  MoveL 1954 to (322.8, 56.16, -151.37) mm, rotated rx -179.9 ry 0 rz -90 deg; joints [37.248, -66.49, 102.161, -126.692, 48.997, 139.557]
  MoveL 1955 to (320.86, 56.08, -150.36) mm, rotated rx -179.9 ry 0 rz -90 deg; joints [37.212, -66.609, 102.338, -126.77, 49.008, 139.643]
  MoveL 1956 to (318.69, 56.01, -150.1) mm, rotated rx -179.9 ry 0 rz -90 deg; joints [37.149, -66.699, 102.475, -126.865, 48.995, 139.733]
  MoveL 1957 to (316.57, 55.93, -150.63) mm, rotated rx -179.9 ry 0 rz -90 deg; joints [37.069, -66.749, 102.554, -126.966, 48.961, 139.816]
  MoveL 1958 to (314.78, 55.85, -151.88) mm, rotated rx -179.9 ry 0 rz -90 deg; joints [36.982, -66.751, 102.565, -127.061, 48.91, 139.882]
  MoveL 1959 to (313.55, 55.78, -153.69) mm, rotated rx -179.9 ry 0 rz -90 deg; joints [36.899, -66.705, 102.507, -127.136, 48.849, 139.923]
  MoveL 1960 to (313.04, 55.7, -155.81) mm, rotated rx -179.9 ry 0 rz -90 deg; joints [36.832, -66.617, 102.388, -127.182, 48.787, 139.933]
  MoveL 1961 to (313.33, 55.62, -157.98) mm, rotated rx -179.9 ry 0 rz -90 deg; joints [36.789, -66.498, 102.224, -127.194, 48.732, 139.913]
  MoveL 1962 to (314.37, 55.55, -159.9) mm, rotated rx -179.9 ry 0 rz -90 deg; joints [36.777, -66.364, 102.036, -127.17, 48.692, 139.866]
  MoveL 1963 to (316.03, 55.47, -161.33) mm, rotated rx -179.9 ry 0 rz -90 deg; joints [36.795, -66.231, 101.851, -127.114, 48.672, 139.797]
  MoveL 1964 to (318.09, 55.39, -162.07) mm, rotated rx -179.9 ry 0 rz -90 deg; joints [36.843, -66.118, 101.691, -127.033, 48.675, 139.717]
  MoveL 1965 to (320.27, 55.32, -162.03) mm, rotated rx -179.9 ry 0 rz -90 deg; joints [36.913, -66.038, 101.58, -126.94, 48.702, 139.638]
  MoveL 1966 to (322.3, 55.24, -161.21) mm, rotated rx -179.9 ry 0 rz -90 deg; joints [36.997, -66.001, 101.531, -126.847, 48.749, 139.571]
  MoveL 1967 to (323.9, 55.16, -159.73) mm, rotated rx -179.9 ry 0 rz -90 deg; joints [37.083, -66.013, 101.552, -126.766, 48.811, 139.524]
  MoveL 1968 to (324.87, 55.09, -157.77) mm, rotated rx -179.9 ry 0 rz -90 deg; joints [37.161, -66.071, 101.64, -126.709, 48.879, 139.506]
  MoveL 1969 to (325.08, 55.01, -155.59) mm, rotated rx -179.9 ry 0 rz -90 deg; joints [37.219, -66.168, 101.784, -126.683, 48.946, 139.518]
  MoveL 1970 to (324.49, 54.93, -153.48) mm, rotated rx -179.9 ry 0 rz -90 deg; joints [37.252, -66.29, 101.965, -126.692, 49.002, 139.56]
  MoveL 1971 to (323.2, 54.86, -151.72) mm, rotated rx -179.9 ry 0 rz -90 deg; joints [37.253, -66.421, 102.16, -126.735, 49.041, 139.627]
  MoveL 1972 to (321.36, 54.78, -150.54) mm, rotated rx -179.9 ry 0 rz -90 deg; joints [37.224, -66.544, 102.344, -126.807, 49.058, 139.71]
  MoveL 1973 to (319.22, 54.7, -150.09) mm, rotated rx -179.9 ry 0 rz -90 deg; joints [37.167, -66.643, 102.493, -126.899, 49.051, 139.8]
  MoveL 1974 to (317.06, 54.63, -150.43) mm, rotated rx -179.9 ry 0 rz -90 deg; joints [37.09, -66.703, 102.587, -127, 49.022, 139.886]
  MoveL 1975 to (315.17, 54.55, -151.52) mm, rotated rx -179.9 ry 0 rz -90 deg; joints [37.004, -66.717, 102.615, -127.097, 48.975, 139.956]
  MoveL 1976 to (313.78, 54.47, -153.21) mm, rotated rx -179.9 ry 0 rz -90 deg; joints [36.919, -66.682, 102.573, -127.178, 48.916, 140.004]
  MoveL 1977 to (313.09, 54.4, -155.28) mm, rotated rx -179.9 ry 0 rz -90 deg; joints [36.847, -66.604, 102.468, -127.232, 48.853, 140.022]
  MoveL 1978 to (313.19, 54.32, -157.47) mm, rotated rx -179.9 ry 0 rz -90 deg; joints [36.798, -66.491, 102.313, -127.252, 48.796, 140.009]
  MoveL 1979 to (314.06, 54.24, -159.47) mm, rotated rx -179.9 ry 0 rz -90 deg; joints [36.778, -66.359, 102.129, -127.237, 48.751, 139.968]
  MoveL 1980 to (315.58, 54.16, -161.04) mm, rotated rx -179.9 ry 0 rz -90 deg; joints [36.789, -66.224, 101.94, -127.188, 48.726, 139.903]
  MoveL 1981 to (317.56, 54.09, -161.96) mm, rotated rx -179.9 ry 0 rz -90 deg; joints [36.83, -66.105, 101.772, -127.112, 48.723, 139.826]
  MoveL 1982 to (319.74, 54.01, -162.11) mm, rotated rx -179.9 ry 0 rz -90 deg; joints [36.895, -66.016, 101.648, -127.021, 48.744, 139.745]
  MoveL 1983 to (321.84, 53.93, -161.48) mm, rotated rx -179.9 ry 0 rz -90 deg; joints [36.977, -65.968, 101.583, -126.927, 48.787, 139.674]
  MoveL 1984 to (323.57, 53.86, -160.14) mm, rotated rx -179.9 ry 0 rz -90 deg; joints [37.063, -65.968, 101.587, -126.842, 48.845, 139.622]
  MoveL 1985 to (324.7, 53.78, -158.27) mm, rotated rx -179.9 ry 0 rz -90 deg; joints [37.144, -66.016, 101.659, -126.778, 48.913, 139.596]
  MoveL 1986 to (325.1, 53.7, -156.12) mm, rotated rx -179.9 ry 0 rz -90 deg; joints [37.208, -66.104, 101.791, -126.744, 48.981, 139.601]
  MoveL 1987 to (324.71, 53.63, -153.97) mm, rotated rx -179.9 ry 0 rz -90 deg; joints [37.247, -66.221, 101.965, -126.744, 49.04, 139.636]
  MoveL 1988 to (323.57, 53.55, -152.1) mm, rotated rx -179.9 ry 0 rz -90 deg; joints [37.256, -66.352, 102.159, -126.779, 49.084, 139.698]
  MoveL 1989 to (321.85, 53.47, -150.76) mm, rotated rx -179.9 ry 0 rz -90 deg; joints [37.234, -66.478, 102.348, -126.845, 49.107, 139.778]
  MoveL 1990 to (319.75, 53.4, -150.12) mm, rotated rx -179.9 ry 0 rz -90 deg; joints [37.183, -66.584, 102.507, -126.933, 49.106, 139.867]
  MoveL 1991 to (317.57, 53.32, -150.27) mm, rotated rx -179.9 ry 0 rz -90 deg; joints [37.111, -66.654, 102.616, -127.033, 49.082, 139.954]
  MoveL 1992 to (315.59, 53.24, -151.19) mm, rotated rx -179.9 ry 0 rz -90 deg; joints [37.025, -66.68, 102.66, -127.132, 49.039, 140.03]
  MoveL 1993 to (314.06, 53.17, -152.75) mm, rotated rx -179.9 ry 0 rz -90 deg; joints [36.939, -66.657, 102.635, -127.218, 48.982, 140.083]
  MoveL 1994 to (313.19, 53.09, -154.76) mm, rotated rx -179.9 ry 0 rz -90 deg; joints [36.863, -66.588, 102.544, -127.279, 48.919, 140.109]
  MoveL 1995 to (313.09, 53.01, -156.94) mm, rotated rx -179.9 ry 0 rz -90 deg; joints [36.808, -66.483, 102.4, -127.308, 48.86, 140.104]
  MoveL 1996 to (313.78, 52.94, -159.02) mm, rotated rx -179.9 ry 0 rz -90 deg; joints [36.78, -66.354, 102.22, -127.302, 48.812, 140.069]
  MoveL 1997 to (315.16, 52.86, -160.71) mm, rotated rx -179.9 ry 0 rz -90 deg; joints [36.784, -66.218, 102.031, -127.26, 48.781, 140.009]
  MoveL 1998 to (317.05, 52.78, -161.8) mm, rotated rx -179.9 ry 0 rz -90 deg; joints [36.818, -66.094, 101.856, -127.19, 48.773, 139.933]
  MoveL 1999 to (319.21, 52.71, -162.15) mm, rotated rx -179.9 ry 0 rz -90 deg; joints [36.878, -65.996, 101.719, -127.102, 48.788, 139.853]
  MoveL 2000 to (321.35, 52.63, -161.7) mm, rotated rx -179.9 ry 0 rz -90 deg; joints [36.957, -65.938, 101.638, -127.007, 48.825, 139.778]
  MoveL 2001 to (323.19, 52.55, -160.52) mm, rotated rx -179.9 ry 0 rz -90 deg; joints [37.043, -65.926, 101.625, -126.919, 48.881, 139.72]
  MoveL 2002 to (324.49, 52.48, -158.76) mm, rotated rx -179.9 ry 0 rz -90 deg; joints [37.126, -65.962, 101.681, -126.849, 48.947, 139.688]
  MoveL 2003 to (325.08, 52.4, -156.65) mm, rotated rx -179.9 ry 0 rz -90 deg; joints [37.195, -66.041, 101.8, -126.807, 49.015, 139.685]
  MoveL 2004 to (324.87, 52.32, -154.48) mm, rotated rx -179.9 ry 0 rz -90 deg; joints [37.241, -66.153, 101.966, -126.799, 49.078, 139.714]
  MoveL 2005 to (323.91, 52.25, -152.52) mm, rotated rx -179.9 ry 0 rz -90 deg; joints [37.258, -66.282, 102.158, -126.825, 49.126, 139.769]
  MoveL 2006 to (322.31, 52.17, -151.03) mm, rotated rx -179.9 ry 0 rz -90 deg; joints [37.243, -66.411, 102.35, -126.884, 49.154, 139.845]
  MoveL 2007 to (320.28, 52.09, -150.21) mm, rotated rx -179.9 ry 0 rz -90 deg; joints [37.199, -66.523, 102.518, -126.967, 49.159, 139.933]
  MoveL 2008 to (318.09, 52.02, -150.16) mm, rotated rx -179.9 ry 0 rz -90 deg; joints [37.13, -66.603, 102.641, -127.065, 49.141, 140.022]
  MoveL 2009 to (316.04, 51.94, -150.9) mm, rotated rx -179.9 ry 0 rz -90 deg; joints [37.047, -66.64, 102.702, -127.166, 49.102, 140.101]
  MoveL 2010 to (314.38, 51.86, -152.32) mm, rotated rx -179.9 ry 0 rz -90 deg; joints [36.96, -66.629, 102.693, -127.256, 49.048, 140.161]
  MoveL 2011 to (313.33, 51.79, -154.25) mm, rotated rx -179.9 ry 0 rz -90 deg; joints [36.881, -66.57, 102.618, -127.325, 48.986, 140.194]
  MoveL 2012 to (313.04, 51.71, -156.41) mm, rotated rx -179.9 ry 0 rz -90 deg; joints [36.82, -66.473, 102.484, -127.362, 48.925, 140.196]
  MoveL 2013 to (313.54, 51.63, -158.54) mm, rotated rx -179.9 ry 0 rz -90 deg; joints [36.785, -66.348, 102.312, -127.364, 48.873, 140.168]
  MoveL 2014 to (314.77, 51.56, -160.35) mm, rotated rx -179.9 ry 0 rz -90 deg; joints [36.781, -66.213, 102.122, -127.331, 48.838, 140.113]
  MoveL 2015 to (316.56, 51.48, -161.6) mm, rotated rx -179.9 ry 0 rz -90 deg; joints [36.808, -66.084, 101.941, -127.267, 48.824, 140.041]
  MoveL 2016 to (318.68, 51.4, -162.14) mm, rotated rx -179.9 ry 0 rz -90 deg; joints [36.862, -65.979, 101.793, -127.182, 48.833, 139.96]
  MoveL 2017 to (320.85, 51.32, -161.88) mm, rotated rx -179.9 ry 0 rz -90 deg; joints [36.937, -65.91, 101.698, -127.088, 48.865, 139.883]
  MoveL 2018 to (322.79, 51.25, -160.87) mm, rotated rx -179.9 ry 0 rz -90 deg; joints [37.023, -65.887, 101.668, -126.997, 48.917, 139.821]
  MoveL 2019 to (324.24, 51.17, -159.23) mm, rotated rx -179.9 ry 0 rz -90 deg; joints [37.107, -65.911, 101.707, -126.921, 48.981, 139.781]
  MoveL 2020 to (325.01, 51.09, -157.18) mm, rotated rx -179.9 ry 0 rz -90 deg; joints [37.181, -65.981, 101.812, -126.872, 49.049, 139.771]
  MoveL 2021 to (325, 51.02, -155) mm, rotated rx -179.9 ry 0 rz -90 deg; joints [37.233, -66.086, 101.968, -126.855, 49.114, 139.792]
  MoveL 2022 to (324.21, 50.94, -152.96) mm, rotated rx -179.9 ry 0 rz -90 deg; joints [37.257, -66.212, 102.156, -126.873, 49.167, 139.842]
  MoveL 2023 to (322.74, 50.86, -151.33) mm, rotated rx -179.9 ry 0 rz -90 deg; joints [37.25, -66.342, 102.35, -126.924, 49.2, 139.914]
  MoveL 2024 to (320.8, 50.79, -150.34) mm, rotated rx -179.9 ry 0 rz -90 deg; joints [37.213, -66.46, 102.526, -127.002, 49.211, 140]
  MoveL 2025 to (318.62, 50.71, -150.1) mm, rotated rx -179.9 ry 0 rz -90 deg; joints [37.149, -66.549, 102.662, -127.098, 49.199, 140.089]
  MoveL 2026 to (316.51, 50.63, -150.65) mm, rotated rx -179.9 ry 0 rz -90 deg; joints [37.069, -66.597, 102.739, -127.199, 49.164, 140.172]
  MoveL 2027 to (314.73, 50.56, -151.93) mm, rotated rx -179.9 ry 0 rz -90 deg; joints [36.982, -66.597, 102.748, -127.293, 49.113, 140.237]
  MoveL 2028 to (313.52, 50.48, -153.75) mm, rotated rx -179.9 ry 0 rz -90 deg; joints [36.899, -66.55, 102.687, -127.368, 49.053, 140.276]
  MoveL 2029 to (313.04, 50.4, -155.88) mm, rotated rx -179.9 ry 0 rz -90 deg; joints [36.833, -66.461, 102.567, -127.414, 48.991, 140.286]
  MoveL 2030 to (313.35, 50.33, -158.04) mm, rotated rx -179.9 ry 0 rz -90 deg; joints [36.791, -66.342, 102.401, -127.424, 48.936, 140.265]
  MoveL 2031 to (314.41, 50.25, -159.95) mm, rotated rx -179.9 ry 0 rz -90 deg; joints [36.78, -66.207, 102.214, -127.399, 48.896, 140.217]
  MoveL 2032 to (316.09, 50.17, -161.36) mm, rotated rx -179.9 ry 0 rz -90 deg; joints [36.799, -66.076, 102.028, -127.342, 48.876, 140.147]
  MoveL 2033 to (318.15, 50.1, -162.08) mm, rotated rx -179.9 ry 0 rz -90 deg; joints [36.848, -65.963, 101.87, -127.262, 48.88, 140.068]
  MoveL 2034 to (320.34, 50.02, -162.02) mm, rotated rx -179.9 ry 0 rz -90 deg; joints [36.918, -65.885, 101.761, -127.168, 48.906, 139.989]
  MoveL 2035 to (322.36, 49.94, -161.18) mm, rotated rx -179.9 ry 0 rz -90 deg; joints [37.002, -65.85, 101.714, -127.075, 48.953, 139.922]
  MoveL 2036 to (323.94, 49.87, -159.67) mm, rotated rx -179.9 ry 0 rz -90 deg; joints [37.088, -65.863, 101.737, -126.995, 49.015, 139.876]
  MoveL 2037 to (324.89, 49.79, -157.7) mm, rotated rx -179.9 ry 0 rz -90 deg; joints [37.165, -65.922, 101.827, -126.938, 49.083, 139.859]
  MoveL 2038 to (325.07, 49.71, -155.52) mm, rotated rx -179.9 ry 0 rz -90 deg; joints [37.223, -66.02, 101.972, -126.913, 49.15, 139.873]
  MoveL 2039 to (324.47, 49.64, -153.42) mm, rotated rx -179.9 ry 0 rz -90 deg; joints [37.255, -66.142, 102.154, -126.922, 49.206, 139.915]
  MoveL 2040 to (323.15, 49.56, -151.68) mm, rotated rx -179.9 ry 0 rz -90 deg; joints [37.256, -66.273, 102.349, -126.966, 49.245, 139.983]
  MoveL 2041 to (321.3, 49.48, -150.51) mm, rotated rx -179.9 ry 0 rz -90 deg; joints [37.225, -66.395, 102.532, -127.039, 49.262, 140.066]
  MoveL 2042 to (319.16, 49.41, -150.09) mm, rotated rx -179.9 ry 0 rz -90 deg; joints [37.167, -66.492, 102.679, -127.131, 49.255, 140.156]
  MoveL 2043 to (317, 49.33, -150.45) mm, rotated rx -179.9 ry 0 rz -90 deg; joints [37.09, -66.551, 102.772, -127.232, 49.226, 140.241]
  MoveL 2044 to (315.12, 49.25, -151.56) mm, rotated rx -179.9 ry 0 rz -90 deg; joints [37.004, -66.563, 102.797, -127.329, 49.178, 140.311]
  MoveL 2045 to (313.75, 49.18, -153.27) mm, rotated rx -179.9 ry 0 rz -90 deg; joints [36.919, -66.527, 102.754, -127.409, 49.119, 140.357]
  MoveL 2046 to (313.08, 49.1, -155.35) mm, rotated rx -179.9 ry 0 rz -90 deg; joints [36.848, -66.448, 102.646, -127.463, 49.057, 140.375]
  MoveL 2047 to (313.2, 49.02, -157.53) mm, rotated rx -179.9 ry 0 rz -90 deg; joints [36.799, -66.334, 102.49, -127.482, 49, 140.361]
  MoveL 2048 to (314.09, 48.94, -159.53) mm, rotated rx -179.9 ry 0 rz -90 deg; joints [36.78, -66.202, 102.305, -127.466, 48.955, 140.318]
  MoveL 2049 to (315.64, 48.87, -161.08) mm, rotated rx -179.9 ry 0 rz -90 deg; joints [36.792, -66.068, 102.117, -127.416, 48.93, 140.253]
  MoveL 2050 to (317.63, 48.79, -161.98) mm, rotated rx -179.9 ry 0 rz -90 deg; joints [36.834, -65.95, 101.95, -127.34, 48.928, 140.175]
  MoveL 2051 to (319.81, 48.71, -162.1) mm, rotated rx -179.9 ry 0 rz -90 deg; joints [36.9, -65.862, 101.827, -127.249, 48.949, 140.095]
  MoveL 2052 to (321.9, 48.64, -161.45) mm, rotated rx -179.9 ry 0 rz -90 deg; joints [36.982, -65.816, 101.764, -127.154, 48.991, 140.024]
  MoveL 2053 to (323.61, 48.56, -160.09) mm, rotated rx -179.9 ry 0 rz -90 deg; joints [37.068, -65.817, 101.77, -127.07, 49.05, 139.973]
  MoveL 2054 to (324.73, 48.48, -158.21) mm, rotated rx -179.9 ry 0 rz -90 deg; joints [37.149, -65.866, 101.845, -127.006, 49.117, 139.948]
  MoveL 2055 to (325.1, 48.41, -156.06) mm, rotated rx -179.9 ry 0 rz -90 deg; joints [37.212, -65.955, 101.978, -126.973, 49.185, 139.954]
  MoveL 2056 to (324.68, 48.33, -153.91) mm, rotated rx -179.9 ry 0 rz -90 deg; joints [37.251, -66.073, 102.153, -126.974, 49.245, 139.99]
  MoveL 2057 to (323.53, 48.25, -152.05) mm, rotated rx -179.9 ry 0 rz -90 deg; joints [37.259, -66.203, 102.348, -127.01, 49.288, 140.052]
  MoveL 2058 to (321.79, 48.18, -150.73) mm, rotated rx -179.9 ry 0 rz -90 deg; joints [37.236, -66.329, 102.536, -127.076, 49.311, 140.133]
  MoveL 2059 to (319.69, 48.1, -150.12) mm, rotated rx -179.9 ry 0 rz -90 deg; joints [37.184, -66.433, 102.693, -127.164, 49.31, 140.222]
  MoveL 2060 to (317.51, 48.02, -150.29) mm, rotated rx -179.9 ry 0 rz -90 deg; joints [37.111, -66.502, 102.8, -127.265, 49.286, 140.309]
  MoveL 2061 to (315.53, 47.95, -151.23) mm, rotated rx -179.9 ry 0 rz -90 deg; joints [37.025, -66.526, 102.843, -127.364, 49.242, 140.384]
  MoveL 2062 to (314.02, 47.87, -152.81) mm, rotated rx -179.9 ry 0 rz -90 deg; joints [36.939, -66.502, 102.816, -127.449, 49.185, 140.436]
  MoveL 2063 to (313.18, 47.79, -154.82) mm, rotated rx -179.9 ry 0 rz -90 deg; joints [36.864, -66.432, 102.723, -127.51, 49.123, 140.461]
  MoveL 2064 to (313.1, 47.72, -157.01) mm, rotated rx -179.9 ry 0 rz -90 deg; joints [36.809, -66.326, 102.577, -127.538, 49.064, 140.455]
  MoveL 2065 to (313.81, 47.64, -159.08) mm, rotated rx -179.9 ry 0 rz -90 deg; joints [36.783, -66.197, 102.397, -127.53, 49.016, 140.419]
  MoveL 2066 to (315.21, 47.56, -160.76) mm, rotated rx -179.9 ry 0 rz -90 deg; joints [36.787, -66.061, 102.207, -127.488, 48.986, 140.358]
  MoveL 2067 to (317.12, 47.49, -161.83) mm, rotated rx -179.9 ry 0 rz -90 deg; joints [36.822, -65.938, 102.033, -127.418, 48.977, 140.282]
  MoveL 2068 to (319.28, 47.41, -162.15) mm, rotated rx -179.9 ry 0 rz -90 deg; joints [36.883, -65.841, 101.897, -127.329, 48.993, 140.202]
  MoveL 2069 to (321.42, 47.33, -161.67) mm, rotated rx -179.9 ry 0 rz -90 deg; joints [36.962, -65.784, 101.819, -127.234, 49.03, 140.128]
  MoveL 2070 to (323.24, 47.26, -160.47) mm, rotated rx -179.9 ry 0 rz -90 deg; joints [37.048, -65.774, 101.808, -127.146, 49.085, 140.071]
  MoveL 2071 to (324.52, 47.18, -158.7) mm, rotated rx -179.9 ry 0 rz -90 deg; joints [37.131, -65.812, 101.866, -127.076, 49.151, 140.039]
  MoveL 2072 to (325.08, 47.1, -156.59) mm, rotated rx -179.9 ry 0 rz -90 deg; joints [37.2, -65.892, 101.987, -127.035, 49.22, 140.038]
  MoveL 2073 to (324.85, 47.03, -154.41) mm, rotated rx -179.9 ry 0 rz -90 deg; joints [37.245, -66.004, 102.154, -127.027, 49.282, 140.067]
  MoveL 2074 to (323.87, 46.95, -152.46) mm, rotated rx -179.9 ry 0 rz -90 deg; joints [37.261, -66.133, 102.345, -127.055, 49.33, 140.123]
  MoveL 2075 to (322.25, 46.87, -150.99) mm, rotated rx -179.9 ry 0 rz -90 deg; joints [37.245, -66.261, 102.537, -127.114, 49.359, 140.2]
  MoveL 2076 to (320.21, 46.8, -150.19) mm, rotated rx -179.9 ry 0 rz -90 deg; joints [37.2, -66.372, 102.705, -127.198, 49.363, 140.288]
  MoveL 2077 to (318.03, 46.72, -150.18) mm, rotated rx -179.9 ry 0 rz -90 deg; joints [37.131, -66.451, 102.825, -127.297, 49.345, 140.377]
  MoveL 2078 to (315.98, 46.64, -150.94) mm, rotated rx -179.9 ry 0 rz -90 deg; joints [37.047, -66.486, 102.884, -127.397, 49.306, 140.455]
  MoveL 2079 to (314.34, 46.57, -152.38) mm, rotated rx -179.9 ry 0 rz -90 deg; joints [36.96, -66.473, 102.874, -127.487, 49.252, 140.514]
  MoveL 2080 to (313.31, 46.49, -154.31) mm, rotated rx -179.9 ry 0 rz -90 deg; joints [36.881, -66.414, 102.796, -127.555, 49.19, 140.545]
  MoveL 2081 to (313.05, 46.41, -156.48) mm, rotated rx -179.9 ry 0 rz -90 deg; joints [36.821, -66.315, 102.661, -127.591, 49.129, 140.547]
  MoveL 2082 to (313.57, 46.33, -158.6) mm, rotated rx -179.9 ry 0 rz -90 deg; joints [36.787, -66.19, 102.487, -127.592, 49.078, 140.517]
  MoveL 2083 to (314.82, 46.26, -160.4) mm, rotated rx -179.9 ry 0 rz -90 deg; joints [36.784, -66.055, 102.298, -127.558, 49.042, 140.462]
  MoveL 2084 to (316.62, 46.18, -161.63) mm, rotated rx -179.9 ry 0 rz -90 deg; joints [36.812, -65.927, 102.118, -127.494, 49.028, 140.389]
  MoveL 2085 to (318.75, 46.1, -162.14) mm, rotated rx -179.9 ry 0 rz -90 deg; joints [36.867, -65.823, 101.971, -127.408, 49.038, 140.309]
  MoveL 2086 to (320.92, 46.03, -161.86) mm, rotated rx -179.9 ry 0 rz -90 deg; joints [36.942, -65.756, 101.877, -127.314, 49.07, 140.232]
  MoveL 2087 to (322.84, 45.95, -160.82) mm, rotated rx -179.9 ry 0 rz -90 deg; joints [37.028, -65.734, 101.849, -127.223, 49.122, 140.17]
  MoveL 2088 to (324.27, 45.87, -159.17) mm, rotated rx -179.9 ry 0 rz -90 deg; joints [37.113, -65.76, 101.891, -127.148, 49.186, 140.132]
  MoveL 2089 to (325.02, 45.8, -157.12) mm, rotated rx -179.9 ry 0 rz -90 deg; joints [37.185, -65.831, 101.998, -127.099, 49.254, 140.123]
  MoveL 2090 to (324.98, 45.72, -154.93) mm, rotated rx -179.9 ry 0 rz -90 deg; joints [37.237, -65.936, 102.155, -127.083, 49.319, 140.145]
  MoveL 2091 to (324.17, 45.64, -152.9) mm, rotated rx -179.9 ry 0 rz -90 deg; joints [37.26, -66.062, 102.343, -127.102, 49.371, 140.195]
  MoveL 2092 to (322.69, 45.57, -151.29) mm, rotated rx -179.9 ry 0 rz -90 deg; joints [37.252, -66.192, 102.537, -127.154, 49.405, 140.267]
  MoveL 2093 to (320.73, 45.49, -150.32) mm, rotated rx -179.9 ry 0 rz -90 deg; joints [37.214, -66.309, 102.713, -127.233, 49.416, 140.354]
  MoveL 2094 to (318.56, 45.41, -150.11) mm, rotated rx -179.9 ry 0 rz -90 deg; joints [37.15, -66.396, 102.846, -127.329, 49.403, 140.443]
  MoveL 2095 to (316.45, 45.34, -150.68) mm, rotated rx -179.9 ry 0 rz -90 deg; joints [37.069, -66.443, 102.921, -127.43, 49.368, 140.525]
  MoveL 2096 to (314.68, 45.26, -151.97) mm, rotated rx -179.9 ry 0 rz -90 deg; joints [36.982, -66.442, 102.928, -127.524, 49.317, 140.589]
  MoveL 2097 to (313.49, 45.18, -153.81) mm, rotated rx -179.9 ry 0 rz -90 deg; joints [36.9, -66.393, 102.866, -127.598, 49.257, 140.628]
  MoveL 2098 to (313.04, 45.11, -155.95) mm, rotated rx -179.9 ry 0 rz -90 deg; joints [36.834, -66.303, 102.743, -127.642, 49.195, 140.637]
  MoveL 2099 to (313.37, 45.03, -158.11) mm, rotated rx -179.9 ry 0 rz -90 deg; joints [36.793, -66.184, 102.577, -127.652, 49.141, 140.614]
  MoveL 2100 to (314.46, 44.95, -160.01) mm, rotated rx -179.9 ry 0 rz -90 deg; joints [36.782, -66.049, 102.389, -127.626, 49.101, 140.565]
  MoveL 2101 to (316.15, 44.88, -161.39) mm, rotated rx -179.9 ry 0 rz -90 deg; joints [36.803, -65.918, 102.204, -127.569, 49.081, 140.495]
  MoveL 2102 to (318.22, 44.8, -162.09) mm, rotated rx -179.9 ry 0 rz -90 deg; joints [36.852, -65.807, 102.047, -127.487, 49.085, 140.416]
  MoveL 2103 to (320.4, 44.72, -162) mm, rotated rx -179.9 ry 0 rz -90 deg; joints [36.923, -65.73, 101.939, -127.393, 49.112, 140.337]
  MoveL 2104 to (322.41, 44.65, -161.14) mm, rotated rx -179.9 ry 0 rz -90 deg; joints [37.008, -65.696, 101.895, -127.3, 49.159, 140.271]
  MoveL 2105 to (323.98, 44.57, -159.62) mm, rotated rx -179.9 ry 0 rz -90 deg; joints [37.093, -65.711, 101.92, -127.221, 49.22, 140.226]
  MoveL 2106 to (324.91, 44.49, -157.64) mm, rotated rx -179.9 ry 0 rz -90 deg; joints [37.17, -65.772, 102.011, -127.165, 49.288, 140.21]
  MoveL 2107 to (325.06, 44.42, -155.46) mm, rotated rx -179.9 ry 0 rz -90 deg; joints [37.228, -65.869, 102.158, -127.14, 49.355, 140.224]
  MoveL 2108 to (324.43, 44.34, -153.36) mm, rotated rx -179.9 ry 0 rz -90 deg; joints [37.258, -65.992, 102.341, -127.15, 49.411, 140.268]
  MoveL 2109 to (323.1, 44.26, -151.63) mm, rotated rx -179.9 ry 0 rz -90 deg; joints [37.258, -66.123, 102.536, -127.195, 49.45, 140.336]
  MoveL 2110 to (321.24, 44.19, -150.49) mm, rotated rx -179.9 ry 0 rz -90 deg; joints [37.226, -66.244, 102.718, -127.268, 49.466, 140.42]
  MoveL 2111 to (319.09, 44.11, -150.09) mm, rotated rx -179.9 ry 0 rz -90 deg; joints [37.168, -66.34, 102.864, -127.361, 49.459, 140.509]
  MoveL 2112 to (316.94, 44.03, -150.47) mm, rotated rx -179.9 ry 0 rz -90 deg; joints [37.09, -66.397, 102.954, -127.462, 49.43, 140.594]
  MoveL 2113 to (315.07, 43.96, -151.6) mm, rotated rx -179.9 ry 0 rz -90 deg; joints [37.004, -66.408, 102.978, -127.559, 49.382, 140.663]
  MoveL 2114 to (313.72, 43.88, -153.33) mm, rotated rx -179.9 ry 0 rz -90 deg; joints [36.919, -66.37, 102.932, -127.639, 49.323, 140.708]
  MoveL 2115 to (313.08, 43.8, -155.42) mm, rotated rx -179.9 ry 0 rz -90 deg; joints [36.849, -66.29, 102.823, -127.691, 49.261, 140.725]
  MoveL 2116 to (313.22, 43.72, -157.6) mm, rotated rx -179.9 ry 0 rz -90 deg; joints [36.801, -66.176, 102.665, -127.71, 49.204, 140.71]
  MoveL 2117 to (314.13, 43.65, -159.58) mm, rotated rx -179.9 ry 0 rz -90 deg; joints [36.783, -66.043, 102.48, -127.692, 49.16, 140.666]
  MoveL 2118 to (315.69, 43.57, -161.12) mm, rotated rx -179.9 ry 0 rz -90 deg; joints [36.796, -65.91, 102.292, -127.642, 49.135, 140.601]
  MoveL 2119 to (317.69, 43.49, -161.99) mm, rotated rx -179.9 ry 0 rz -90 deg; joints [36.839, -65.793, 102.126, -127.565, 49.133, 140.522]
  MoveL 2120 to (319.88, 43.42, -162.1) mm, rotated rx -179.9 ry 0 rz -90 deg; joints [36.905, -65.706, 102.005, -127.473, 49.154, 140.442]
  MoveL 2121 to (321.96, 43.34, -161.41) mm, rotated rx -179.9 ry 0 rz -90 deg; joints [36.987, -65.662, 101.944, -127.379, 49.197, 140.372]
  MoveL 2122 to (323.65, 43.26, -160.04) mm, rotated rx -179.9 ry 0 rz -90 deg; joints [37.074, -65.665, 101.952, -127.295, 49.255, 140.322]
  MoveL 2123 to (324.75, 43.19, -158.15) mm, rotated rx -179.9 ry 0 rz -90 deg; joints [37.154, -65.714, 102.028, -127.232, 49.323, 140.298]
  MoveL 2124 to (325.1, 43.11, -155.99) mm, rotated rx -179.9 ry 0 rz -90 deg; joints [37.217, -65.804, 102.163, -127.199, 49.39, 140.305]
  MoveL 2125 to (324.66, 43.03, -153.85) mm, rotated rx -179.9 ry 0 rz -90 deg; joints [37.254, -65.922, 102.339, -127.201, 49.45, 140.342]
  MoveL 2126 to (323.48, 42.96, -152) mm, rotated rx -179.9 ry 0 rz -90 deg; joints [37.261, -66.052, 102.534, -127.237, 49.493, 140.405]
  MoveL 2127 to (321.73, 42.88, -150.7) mm, rotated rx -179.9 ry 0 rz -90 deg; joints [37.237, -66.177, 102.721, -127.304, 49.516, 140.486]
  MoveL 2128 to (319.62, 42.8, -150.11) mm, rotated rx -179.9 ry 0 rz -90 deg; joints [37.185, -66.28, 102.878, -127.393, 49.514, 140.575]
  MoveL 2129 to (317.44, 42.73, -150.31) mm, rotated rx -179.9 ry 0 rz -90 deg; joints [37.111, -66.348, 102.983, -127.494, 49.49, 140.661]
  MoveL 2130 to (315.48, 42.65, -151.27) mm, rotated rx -179.9 ry 0 rz -90 deg; joints [37.025, -66.37, 103.023, -127.593, 49.447, 140.735]
  MoveL 2131 to (313.99, 42.57, -152.87) mm, rotated rx -179.9 ry 0 rz -90 deg; joints [36.94, -66.344, 102.994, -127.678, 49.39, 140.787]
  MoveL 2132 to (313.16, 42.5, -154.89) mm, rotated rx -179.9 ry 0 rz -90 deg; joints [36.865, -66.274, 102.899, -127.738, 49.328, 140.811]
  MoveL 2133 to (313.11, 42.42, -157.08) mm, rotated rx -179.9 ry 0 rz -90 deg; joints [36.811, -66.167, 102.752, -127.765, 49.269, 140.803]
  MoveL 2134 to (313.84, 42.34, -159.14) mm, rotated rx -179.9 ry 0 rz -90 deg; joints [36.785, -66.037, 102.571, -127.756, 49.221, 140.766]
  MoveL 2135 to (315.26, 42.27, -160.8) mm, rotated rx -179.9 ry 0 rz -90 deg; joints [36.79, -65.903, 102.381, -127.713, 49.191, 140.705]
  MoveL 2136 to (317.18, 42.19, -161.85) mm, rotated rx -179.9 ry 0 rz -90 deg; joints [36.826, -65.78, 102.208, -127.642, 49.183, 140.629]
  MoveL 2137 to (319.35, 42.11, -162.14) mm, rotated rx -179.9 ry 0 rz -90 deg; joints [36.888, -65.685, 102.074, -127.553, 49.198, 140.548]
  MoveL 2138 to (321.48, 42.04, -161.65) mm, rotated rx -179.9 ry 0 rz -90 deg; joints [36.967, -65.629, 101.997, -127.458, 49.236, 140.475]
  MoveL 2139 to (323.29, 41.96, -160.43) mm, rotated rx -179.9 ry 0 rz -90 deg; joints [37.054, -65.621, 101.988, -127.37, 49.291, 140.419]
  MoveL 2140 to (324.55, 41.88, -158.64) mm, rotated rx -179.9 ry 0 rz -90 deg; joints [37.136, -65.66, 102.049, -127.301, 49.357, 140.388]
  MoveL 2141 to (325.09, 41.81, -156.52) mm, rotated rx -179.9 ry 0 rz -90 deg; joints [37.204, -65.741, 102.171, -127.26, 49.425, 140.388]
  MoveL 2142 to (324.84, 41.73, -154.35) mm, rotated rx -179.9 ry 0 rz -90 deg; joints [37.248, -65.853, 102.339, -127.254, 49.487, 140.418]
  MoveL 2143 to (323.83, 41.65, -152.41) mm, rotated rx -179.9 ry 0 rz -90 deg; joints [37.263, -65.982, 102.531, -127.282, 49.535, 140.475]
  MoveL 2144 to (322.19, 41.58, -150.96) mm, rotated rx -179.9 ry 0 rz -90 deg; joints [37.247, -66.109, 102.723, -127.342, 49.564, 140.552]
  MoveL 2145 to (320.15, 41.5, -150.18) mm, rotated rx -179.9 ry 0 rz -90 deg; joints [37.201, -66.219, 102.889, -127.426, 49.568, 140.64]
  MoveL 2146 to (317.96, 41.42, -150.19) mm, rotated rx -179.9 ry 0 rz -90 deg; joints [37.131, -66.296, 103.008, -127.525, 49.55, 140.728]
  MoveL 2147 to (315.92, 41.35, -150.97) mm, rotated rx -179.9 ry 0 rz -90 deg; joints [37.047, -66.33, 103.065, -127.626, 49.51, 140.806]
  MoveL 2148 to (314.29, 41.27, -152.43) mm, rotated rx -179.9 ry 0 rz -90 deg; joints [36.96, -66.316, 103.052, -127.715, 49.456, 140.864]
  MoveL 2149 to (313.29, 41.19, -154.37) mm, rotated rx -179.9 ry 0 rz -90 deg; joints [36.882, -66.255, 102.972, -127.782, 49.395, 140.895]
  MoveL 2150 to (313.05, 41.11, -156.55) mm, rotated rx -179.9 ry 0 rz -90 deg; joints [36.822, -66.156, 102.836, -127.818, 49.334, 140.895]
  MoveL 2151 to (313.6, 41.04, -158.66) mm, rotated rx -179.9 ry 0 rz -90 deg; joints [36.789, -66.031, 102.661, -127.818, 49.283, 140.865]
  MoveL 2152 to (314.87, 40.96, -160.45) mm, rotated rx -179.9 ry 0 rz -90 deg; joints [36.787, -65.896, 102.471, -127.783, 49.248, 140.809]
  MoveL 2153 to (316.68, 40.88, -161.66) mm, rotated rx -179.9 ry 0 rz -90 deg; joints [36.816, -65.769, 102.292, -127.718, 49.234, 140.735]
  MoveL 2154 to (318.82, 40.81, -162.14) mm, rotated rx -179.9 ry 0 rz -90 deg; joints [36.872, -65.666, 102.146, -127.632, 49.244, 140.655]
  MoveL 2155 to (320.98, 40.73, -161.84) mm, rotated rx -179.9 ry 0 rz -90 deg; joints [36.948, -65.6, 102.054, -127.537, 49.276, 140.578]
  MoveL 2156 to (322.89, 40.65, -160.78) mm, rotated rx -179.9 ry 0 rz -90 deg; joints [37.033, -65.58, 102.029, -127.446, 49.328, 140.517]
  MoveL 2157 to (324.3, 40.58, -159.11) mm, rotated rx -179.9 ry 0 rz -90 deg; joints [37.118, -65.607, 102.073, -127.372, 49.391, 140.48]
  MoveL 2158 to (325.03, 40.5, -157.05) mm, rotated rx -179.9 ry 0 rz -90 deg; joints [37.19, -65.679, 102.181, -127.323, 49.46, 140.472]
  MoveL 2159 to (324.97, 40.42, -154.86) mm, rotated rx -179.9 ry 0 rz -90 deg; joints [37.241, -65.785, 102.34, -127.308, 49.524, 140.495]
  MoveL 2160 to (324.13, 40.35, -152.84) mm, rotated rx -179.9 ry 0 rz -90 deg; joints [37.263, -65.911, 102.528, -127.328, 49.577, 140.546]
  MoveL 2161 to (322.64, 40.27, -151.25) mm, rotated rx -179.9 ry 0 rz -90 deg; joints [37.254, -66.04, 102.722, -127.381, 49.61, 140.619]
  MoveL 2162 to (320.67, 40.19, -150.3) mm, rotated rx -179.9 ry 0 rz -90 deg; joints [37.215, -66.156, 102.897, -127.46, 49.621, 140.705]
  MoveL 2163 to (318.49, 40.12, -150.11) mm, rotated rx -179.9 ry 0 rz -90 deg; joints [37.15, -66.242, 103.029, -127.556, 49.608, 140.794]
  MoveL 2164 to (316.39, 40.04, -150.71) mm, rotated rx -179.9 ry 0 rz -90 deg; joints [37.069, -66.287, 103.102, -127.658, 49.573, 140.876]
  MoveL 2165 to (314.64, 39.96, -152.02) mm, rotated rx -179.9 ry 0 rz -90 deg; joints [36.982, -66.284, 103.106, -127.751, 49.522, 140.939]
  MoveL 2166 to (313.47, 39.89, -153.87) mm, rotated rx -179.9 ry 0 rz -90 deg; joints [36.9, -66.235, 103.042, -127.825, 49.462, 140.977]
  MoveL 2167 to (313.04, 39.81, -156.01) mm, rotated rx -179.9 ry 0 rz -90 deg; joints [36.835, -66.144, 102.918, -127.869, 49.4, 140.984]
  MoveL 2168 to (313.4, 39.73, -158.17) mm, rotated rx -179.9 ry 0 rz -90 deg; joints [36.795, -66.023, 102.75, -127.877, 49.346, 140.961]
  MoveL 2169 to (314.5, 39.66, -160.06) mm, rotated rx -179.9 ry 0 rz -90 deg; joints [36.785, -65.889, 102.562, -127.851, 49.306, 140.911]
  MoveL 2170 to (316.2, 39.58, -161.43) mm, rotated rx -179.9 ry 0 rz -90 deg; joints [36.807, -65.759, 102.377, -127.792, 49.287, 140.841]
  MoveL 2171 to (318.28, 39.5, -162.1) mm, rotated rx -179.9 ry 0 rz -90 deg; joints [36.857, -65.649, 102.222, -127.71, 49.291, 140.761]
  MoveL 2172 to (320.47, 39.43, -161.99) mm, rotated rx -179.9 ry 0 rz -90 deg; joints [36.929, -65.573, 102.115, -127.616, 49.318, 140.682]
  MoveL 2173 to (322.47, 39.35, -161.1) mm, rotated rx -179.9 ry 0 rz -90 deg; joints [37.013, -65.541, 102.073, -127.523, 49.365, 140.617]
  MoveL 2174 to (324.02, 39.27, -159.56) mm, rotated rx -179.9 ry 0 rz -90 deg; joints [37.099, -65.557, 102.1, -127.444, 49.426, 140.573]
  MoveL 2175 to (324.92, 39.2, -157.57) mm, rotated rx -179.9 ry 0 rz -90 deg; joints [37.175, -65.619, 102.194, -127.388, 49.494, 140.558]
  MoveL 2176 to (325.06, 39.12, -155.39) mm, rotated rx -179.9 ry 0 rz -90 deg; joints [37.232, -65.717, 102.342, -127.365, 49.561, 140.573]
  MoveL 2177 to (324.4, 39.04, -153.3) mm, rotated rx -179.9 ry 0 rz -90 deg; joints [37.261, -65.84, 102.525, -127.376, 49.617, 140.618]
  MoveL 2178 to (323.05, 38.97, -151.59) mm, rotated rx -179.9 ry 0 rz -90 deg; joints [37.26, -65.97, 102.72, -127.421, 49.655, 140.686]
  MoveL 2179 to (321.17, 38.89, -150.46) mm, rotated rx -179.9 ry 0 rz -90 deg; joints [37.228, -66.091, 102.902, -127.495, 49.672, 140.77]
  MoveL 2180 to (319.02, 38.81, -150.09) mm, rotated rx -179.9 ry 0 rz -90 deg; joints [37.169, -66.185, 103.046, -127.588, 49.664, 140.86]
  MoveL 2181 to (316.87, 38.74, -150.5) mm, rotated rx -179.9 ry 0 rz -90 deg; joints [37.09, -66.241, 103.134, -127.689, 49.635, 140.944]
  MoveL 2182 to (315.02, 38.66, -151.65) mm, rotated rx -179.9 ry 0 rz -90 deg; joints [37.004, -66.25, 103.156, -127.786, 49.588, 141.012]
  MoveL 2183 to (313.69, 38.58, -153.39) mm, rotated rx -179.9 ry 0 rz -90 deg; joints [36.92, -66.211, 103.108, -127.865, 49.529, 141.057]
  MoveL 2184 to (313.07, 38.5, -155.48) mm, rotated rx -179.9 ry 0 rz -90 deg; joints [36.85, -66.13, 102.997, -127.917, 49.467, 141.072]
  MoveL 2185 to (313.24, 38.43, -157.66) mm, rotated rx -179.9 ry 0 rz -90 deg; joints [36.803, -66.015, 102.838, -127.935, 49.41, 141.056]
  MoveL 2186 to (314.17, 38.35, -159.64) mm, rotated rx -179.9 ry 0 rz -90 deg; joints [36.785, -65.883, 102.653, -127.916, 49.366, 141.012]
  MoveL 2187 to (315.75, 38.27, -161.15) mm, rotated rx -179.9 ry 0 rz -90 deg; joints [36.799, -65.75, 102.465, -127.865, 49.341, 140.946]
  MoveL 2188 to (317.76, 38.2, -162.01) mm, rotated rx -179.9 ry 0 rz -90 deg; joints [36.843, -65.634, 102.3, -127.788, 49.339, 140.867]
  MoveL 2189 to (319.94, 38.12, -162.09) mm, rotated rx -179.9 ry 0 rz -90 deg; joints [36.91, -65.549, 102.18, -127.695, 49.36, 140.787]
  MoveL 2190 to (322.01, 38.04, -161.38) mm, rotated rx -179.9 ry 0 rz -90 deg; joints [36.992, -65.506, 102.121, -127.601, 49.403, 140.718]
  MoveL 2191 to (323.7, 37.97, -159.99) mm, rotated rx -179.9 ry 0 rz -90 deg; joints [37.079, -65.51, 102.131, -127.517, 49.462, 140.668]
  MoveL 2192 to (324.77, 37.89, -158.08) mm, rotated rx -179.9 ry 0 rz -90 deg; joints [37.159, -65.561, 102.21, -127.455, 49.529, 140.645]
  MoveL 2193 to (325.1, 37.81, -155.92) mm, rotated rx -179.9 ry 0 rz -90 deg; joints [37.221, -65.652, 102.346, -127.423, 49.596, 140.653]
  MoveL 2194 to (324.63, 37.74, -153.78) mm, rotated rx -179.9 ry 0 rz -90 deg; joints [37.257, -65.77, 102.523, -127.425, 49.656, 140.691]
  MoveL 2195 to (323.43, 37.66, -151.96) mm, rotated rx -179.9 ry 0 rz -90 deg; joints [37.264, -65.9, 102.718, -127.463, 49.699, 140.755]
  MoveL 2196 to (321.66, 37.58, -150.67) mm, rotated rx -179.9 ry 0 rz -90 deg; joints [37.239, -66.024, 102.905, -127.53, 49.721, 140.836]
  MoveL 2197 to (319.55, 37.51, -150.1) mm, rotated rx -179.9 ry 0 rz -90 deg; joints [37.186, -66.126, 103.06, -127.62, 49.72, 140.925]
  MoveL 2198 to (317.38, 37.43, -150.33) mm, rotated rx -179.9 ry 0 rz -90 deg; joints [37.111, -66.192, 103.163, -127.72, 49.696, 141.011]
  MoveL 2199 to (315.43, 37.35, -151.31) mm, rotated rx -179.9 ry 0 rz -90 deg; joints [37.025, -66.213, 103.201, -127.819, 49.652, 141.084]
  MoveL 2200 to (313.95, 37.28, -152.92) mm, rotated rx -179.9 ry 0 rz -90 deg; joints [36.94, -66.185, 103.17, -127.904, 49.595, 141.135]
  MoveL 2201 to (313.15, 37.2, -154.96) mm, rotated rx -179.9 ry 0 rz -90 deg; joints [36.865, -66.113, 103.073, -127.963, 49.533, 141.158]
  MoveL 2202 to (313.12, 37.12, -157.14) mm, rotated rx -179.9 ry 0 rz -90 deg; joints [36.812, -66.006, 102.924, -127.989, 49.475, 141.149]
  MoveL 2203 to (313.88, 37.05, -159.19) mm, rotated rx -179.9 ry 0 rz -90 deg; joints [36.787, -65.876, 102.743, -127.98, 49.427, 141.111]
  MoveL 2204 to (315.32, 36.97, -160.84) mm, rotated rx -179.9 ry 0 rz -90 deg; joints [36.794, -65.742, 102.553, -127.936, 49.397, 141.05]
  MoveL 2205 to (317.25, 36.89, -161.87) mm, rotated rx -179.9 ry 0 rz -90 deg; joints [36.831, -65.62, 102.381, -127.864, 49.389, 140.973]
  MoveL 2206 to (319.41, 36.82, -162.14) mm, rotated rx -179.9 ry 0 rz -90 deg; joints [36.893, -65.526, 102.248, -127.774, 49.405, 140.893]
  MoveL 2207 to (321.54, 36.74, -161.62) mm, rotated rx -179.9 ry 0 rz -90 deg; joints [36.972, -65.473, 102.173, -127.679, 49.442, 140.819]
  MoveL 2208 to (323.34, 36.66, -160.38) mm, rotated rx -179.9 ry 0 rz -90 deg; joints [37.059, -65.465, 102.167, -127.592, 49.498, 140.764]
  MoveL 2209 to (324.58, 36.59, -158.58) mm, rotated rx -179.9 ry 0 rz -90 deg; joints [37.141, -65.505, 102.229, -127.523, 49.563, 140.735]
  MoveL 2210 to (325.09, 36.51, -156.45) mm, rotated rx -179.9 ry 0 rz -90 deg; joints [37.208, -65.587, 102.353, -127.483, 49.632, 140.735]
  MoveL 2211 to (324.82, 36.43, -154.28) mm, rotated rx -179.9 ry 0 rz -90 deg; joints [37.252, -65.7, 102.522, -127.477, 49.694, 140.766]
  MoveL 2212 to (323.78, 36.36, -152.36) mm, rotated rx -179.9 ry 0 rz -90 deg; joints [37.266, -65.828, 102.714, -127.506, 49.741, 140.824]
  MoveL 2213 to (322.13, 36.28, -150.92) mm, rotated rx -179.9 ry 0 rz -90 deg; joints [37.248, -65.956, 102.906, -127.567, 49.769, 140.901]
  MoveL 2214 to (320.08, 36.2, -150.17) mm, rotated rx -179.9 ry 0 rz -90 deg; joints [37.201, -66.064, 103.07, -127.652, 49.774, 140.99]
  MoveL 2215 to (317.9, 36.13, -150.2) mm, rotated rx -179.9 ry 0 rz -90 deg; joints [37.131, -66.14, 103.188, -127.751, 49.755, 141.078]
  MoveL 2216 to (315.86, 36.05, -151.01) mm, rotated rx -179.9 ry 0 rz -90 deg; joints [37.047, -66.172, 103.243, -127.852, 49.716, 141.155]
  MoveL 2217 to (314.25, 35.97, -152.48) mm, rotated rx -179.9 ry 0 rz -90 deg; joints [36.961, -66.157, 103.228, -127.941, 49.662, 141.212]
  MoveL 2218 to (313.27, 35.89, -154.44) mm, rotated rx -179.9 ry 0 rz -90 deg; joints [36.882, -66.095, 103.146, -128.007, 49.601, 141.241]
  MoveL 2219 to (313.06, 35.82, -156.61) mm, rotated rx -179.9 ry 0 rz -90 deg; joints [36.823, -65.995, 103.008, -128.042, 49.54, 141.24]
  MoveL 2220 to (313.63, 35.74, -158.72) mm, rotated rx -179.9 ry 0 rz -90 deg; joints [36.791, -65.869, 102.833, -128.041, 49.489, 141.209]
  MoveL 2221 to (314.91, 35.66, -160.49) mm, rotated rx -179.9 ry 0 rz -90 deg; joints [36.79, -65.735, 102.643, -128.005, 49.454, 141.153]
  MoveL 2222 to (316.75, 35.59, -161.68) mm, rotated rx -179.9 ry 0 rz -90 deg; joints [36.82, -65.608, 102.464, -127.939, 49.44, 141.079]
  MoveL 2223 to (318.88, 35.51, -162.15) mm, rotated rx -179.9 ry 0 rz -90 deg; joints [36.876, -65.507, 102.32, -127.853, 49.45, 140.998]
  MoveL 2224 to (321.04, 35.43, -161.82) mm, rotated rx -179.9 ry 0 rz -90 deg; joints [36.953, -65.442, 102.23, -127.758, 49.483, 140.922]
  MoveL 2225 to (322.94, 35.36, -160.74) mm, rotated rx -179.9 ry 0 rz -90 deg; joints [37.039, -65.423, 102.206, -127.667, 49.534, 140.862]
  MoveL 2226 to (324.34, 35.28, -159.05) mm, rotated rx -179.9 ry 0 rz -90 deg; joints [37.123, -65.452, 102.252, -127.593, 49.598, 140.825]
  MoveL 2227 to (325.04, 35.2, -156.98) mm, rotated rx -179.9 ry 0 rz -90 deg; joints [37.195, -65.525, 102.362, -127.545, 49.667, 140.818]
  MoveL 2228 to (324.95, 35.13, -154.8) mm, rotated rx -179.9 ry 0 rz -90 deg; joints [37.245, -65.631, 102.522, -127.531, 49.731, 140.842]
  MoveL 2229 to (324.1, 35.05, -152.79) mm, rotated rx -179.9 ry 0 rz -90 deg; joints [37.266, -65.757, 102.711, -127.551, 49.783, 140.894]
  MoveL 2230 to (322.58, 34.97, -151.21) mm, rotated rx -179.9 ry 0 rz -90 deg; joints [37.256, -65.886, 102.905, -127.605, 49.816, 140.968]
  MoveL 2231 to (320.6, 34.9, -150.28) mm, rotated rx -179.9 ry 0 rz -90 deg; joints [37.216, -66.001, 103.078, -127.685, 49.827, 141.054]
  MoveL 2232 to (318.42, 34.82, -150.12) mm, rotated rx -179.9 ry 0 rz -90 deg; joints [37.151, -66.085, 103.209, -127.782, 49.814, 141.143]
  MoveL 2233 to (316.33, 34.74, -150.74) mm, rotated rx -179.9 ry 0 rz -90 deg; joints [37.069, -66.129, 103.28, -127.883, 49.779, 141.224]
  MoveL 2234 to (314.59, 34.67, -152.07) mm, rotated rx -179.9 ry 0 rz -90 deg; joints [36.982, -66.125, 103.282, -127.976, 49.728, 141.286]
  MoveL 2235 to (313.44, 34.59, -153.93) mm, rotated rx -179.9 ry 0 rz -90 deg; joints [36.901, -66.074, 103.216, -128.049, 49.668, 141.323]
  MoveL 2236 to (313.04, 34.51, -156.08) mm, rotated rx -179.9 ry 0 rz -90 deg; joints [36.836, -65.982, 103.09, -128.092, 49.606, 141.329]
  MoveL 2237 to (313.42, 34.44, -158.23) mm, rotated rx -179.9 ry 0 rz -90 deg; joints [36.797, -65.861, 102.921, -128.1, 49.552, 141.305]
  MoveL 2238 to (314.54, 34.36, -160.11) mm, rotated rx -179.9 ry 0 rz -90 deg; joints [36.788, -65.728, 102.733, -128.072, 49.513, 141.254]
  MoveL 2239 to (316.26, 34.28, -161.46) mm, rotated rx -179.9 ry 0 rz -90 deg; joints [36.811, -65.598, 102.549, -128.013, 49.493, 141.184]
  MoveL 2240 to (318.35, 34.21, -162.11) mm, rotated rx -179.9 ry 0 rz -90 deg; joints [36.861, -65.489, 102.394, -127.93, 49.497, 141.104]
  MoveL 2241 to (320.53, 34.13, -161.97) mm, rotated rx -179.9 ry 0 rz -90 deg; joints [36.934, -65.414, 102.289, -127.836, 49.524, 141.026]
  MoveL 2242 to (322.52, 34.05, -161.06) mm, rotated rx -179.9 ry 0 rz -90 deg; joints [37.018, -65.384, 102.249, -127.743, 49.572, 140.961]
  MoveL 2243 to (324.06, 33.98, -159.51) mm, rotated rx -179.9 ry 0 rz -90 deg; joints [37.104, -65.402, 102.278, -127.664, 49.633, 140.918]
  MoveL 2244 to (324.94, 33.9, -157.51) mm, rotated rx -179.9 ry 0 rz -90 deg; joints [37.18, -65.464, 102.374, -127.609, 49.701, 140.903]
  MoveL 2245 to (325.05, 33.82, -155.32) mm, rotated rx -179.9 ry 0 rz -90 deg; joints [37.236, -65.563, 102.523, -127.586, 49.767, 140.92]
  MoveL 2246 to (324.37, 33.75, -153.24) mm, rotated rx -179.9 ry 0 rz -90 deg; joints [37.264, -65.686, 102.708, -127.599, 49.823, 140.965]
  MoveL 2247 to (323, 33.67, -151.54) mm, rotated rx -179.9 ry 0 rz -90 deg; joints [37.262, -65.816, 102.903, -127.644, 49.861, 141.034]
  MoveL 2248 to (321.11, 33.59, -150.44) mm, rotated rx -179.9 ry 0 rz -90 deg; joints [37.229, -65.935, 103.083, -127.719, 49.878, 141.119]
  MoveL 2249 to (318.95, 33.52, -150.09) mm, rotated rx -179.9 ry 0 rz -90 deg; joints [37.169, -66.029, 103.226, -127.813, 49.871, 141.208]
  MoveL 2250 to (316.81, 33.44, -150.52) mm, rotated rx -179.9 ry 0 rz -90 deg; joints [37.091, -66.083, 103.312, -127.914, 49.841, 141.292]
  MoveL 2251 to (314.97, 33.36, -151.69) mm, rotated rx -179.9 ry 0 rz -90 deg; joints [37.004, -66.09, 103.332, -128.01, 49.794, 141.359]
  MoveL 2252 to (313.66, 33.28, -153.45) mm, rotated rx -179.9 ry 0 rz -90 deg; joints [36.92, -66.05, 103.281, -128.089, 49.735, 141.403]
  MoveL 2253 to (313.06, 33.21, -155.55) mm, rotated rx -179.9 ry 0 rz -90 deg; joints [36.85, -65.968, 103.169, -128.14, 49.673, 141.417]
  MoveL 2254 to (313.25, 33.13, -157.73) mm, rotated rx -179.9 ry 0 rz -90 deg; joints [36.804, -65.853, 103.009, -128.157, 49.616, 141.4]
  MoveL 2255 to (314.21, 33.05, -159.69) mm, rotated rx -179.9 ry 0 rz -90 deg; joints [36.788, -65.721, 102.823, -128.138, 49.572, 141.355]
  MoveL 2256 to (315.8, 32.98, -161.19) mm, rotated rx -179.9 ry 0 rz -90 deg; joints [36.803, -65.588, 102.635, -128.085, 49.548, 141.288]
  MoveL 2257 to (317.83, 32.9, -162.02) mm, rotated rx -179.9 ry 0 rz -90 deg; joints [36.847, -65.473, 102.471, -128.007, 49.546, 141.209]
  MoveL 2258 to (320.01, 32.82, -162.08) mm, rotated rx -179.9 ry 0 rz -90 deg; joints [36.915, -65.389, 102.353, -127.915, 49.567, 141.13]
  MoveL 2259 to (322.07, 32.75, -161.35) mm, rotated rx -179.9 ry 0 rz -90 deg; joints [36.998, -65.348, 102.296, -127.82, 49.61, 141.061]
  MoveL 2260 to (323.74, 32.67, -159.93) mm, rotated rx -179.9 ry 0 rz -90 deg; joints [37.084, -65.353, 102.309, -127.737, 49.669, 141.012]
  MoveL 2261 to (324.79, 32.59, -158.02) mm, rotated rx -179.9 ry 0 rz -90 deg; joints [37.163, -65.406, 102.389, -127.675, 49.736, 140.99]
  MoveL 2262 to (325.09, 32.52, -155.85) mm, rotated rx -179.9 ry 0 rz -90 deg; joints [37.225, -65.497, 102.527, -127.644, 49.803, 140.999]
  MoveL 2263 to (324.61, 32.44, -153.72) mm, rotated rx -179.9 ry 0 rz -90 deg; joints [37.261, -65.615, 102.705, -127.647, 49.862, 141.038]
  MoveL 2264 to (323.39, 32.36, -151.91) mm, rotated rx -179.9 ry 0 rz -90 deg; joints [37.266, -65.745, 102.899, -127.685, 49.905, 141.102]
  MoveL 2265 to (321.6, 32.29, -150.64) mm, rotated rx -179.9 ry 0 rz -90 deg; joints [37.24, -65.868, 103.086, -127.754, 49.928, 141.183]
  MoveL 2266 to (319.49, 32.21, -150.1) mm, rotated rx -179.9 ry 0 rz -90 deg; joints [37.186, -65.969, 103.24, -127.844, 49.926, 141.273]
  MoveL 2267 to (317.31, 32.13, -150.35) mm, rotated rx -179.9 ry 0 rz -90 deg; joints [37.111, -66.034, 103.341, -127.944, 49.902, 141.359]
  MoveL 2268 to (315.37, 32.06, -151.35) mm, rotated rx -179.9 ry 0 rz -90 deg; joints [37.026, -66.053, 103.377, -128.043, 49.858, 141.431]
  MoveL 2269 to (313.92, 31.98, -152.98) mm, rotated rx -179.9 ry 0 rz -90 deg; joints [36.94, -66.024, 103.343, -128.127, 49.802, 141.481]
  MoveL 2270 to (313.14, 31.9, -155.02) mm, rotated rx -179.9 ry 0 rz -90 deg; joints [36.866, -65.951, 103.245, -128.186, 49.74, 141.502]
  MoveL 2271 to (313.13, 31.83, -157.21) mm, rotated rx -179.9 ry 0 rz -90 deg; joints [36.814, -65.843, 103.095, -128.211, 49.681, 141.493]
  MoveL 2272 to (313.91, 31.75, -159.25) mm, rotated rx -179.9 ry 0 rz -90 deg; joints [36.79, -65.713, 102.913, -128.201, 49.634, 141.454]
  MoveL 2273 to (315.37, 31.67, -160.88) mm, rotated rx -179.9 ry 0 rz -90 deg; joints [36.797, -65.58, 102.723, -128.156, 49.604, 141.391]
  MoveL 2274 to (317.31, 31.6, -161.89) mm, rotated rx -179.9 ry 0 rz -90 deg; joints [36.835, -65.459, 102.551, -128.083, 49.596, 141.315]
  MoveL 2275 to (319.48, 31.52, -162.14) mm, rotated rx -179.9 ry 0 rz -90 deg; joints [36.898, -65.366, 102.42, -127.993, 49.612, 141.234]
  MoveL 2276 to (321.6, 31.44, -161.59) mm, rotated rx -179.9 ry 0 rz -90 deg; joints [36.978, -65.314, 102.347, -127.898, 49.65, 141.162]
  MoveL 2277 to (323.38, 31.37, -160.33) mm, rotated rx -179.9 ry 0 rz -90 deg; joints [37.064, -65.308, 102.343, -127.811, 49.705, 141.107]
  MoveL 2278 to (324.6, 31.29, -158.52) mm, rotated rx -179.9 ry 0 rz -90 deg; joints [37.146, -65.349, 102.407, -127.743, 49.771, 141.078]
  MoveL 2279 to (325.09, 31.21, -156.39) mm, rotated rx -179.9 ry 0 rz -90 deg; joints [37.213, -65.432, 102.533, -127.704, 49.839, 141.08]
  MoveL 2280 to (324.79, 31.14, -154.22) mm, rotated rx -179.9 ry 0 rz -90 deg; joints [37.255, -65.545, 102.703, -127.698, 49.901, 141.112]
  MoveL 2281 to (323.74, 31.06, -152.3) mm, rotated rx -179.9 ry 0 rz -90 deg; joints [37.269, -65.674, 102.896, -127.728, 49.948, 141.17]
  MoveL 2282 to (322.08, 30.98, -150.89) mm, rotated rx -179.9 ry 0 rz -90 deg; joints [37.25, -65.8, 103.086, -127.79, 49.976, 141.249]
  MoveL 2283 to (320.02, 30.91, -150.16) mm, rotated rx -179.9 ry 0 rz -90 deg; joints [37.202, -65.907, 103.25, -127.875, 49.98, 141.337]
  MoveL 2284 to (317.83, 30.83, -150.21) mm, rotated rx -179.9 ry 0 rz -90 deg; joints [37.132, -65.982, 103.366, -127.975, 49.962, 141.424]
  MoveL 2285 to (315.81, 30.75, -151.04) mm, rotated rx -179.9 ry 0 rz -90 deg; joints [37.047, -66.012, 103.418, -128.075, 49.922, 141.501]
  MoveL 2286 to (314.21, 30.67, -152.54) mm, rotated rx -179.9 ry 0 rz -90 deg; joints [36.961, -65.995, 103.401, -128.164, 49.868, 141.557]
  MoveL 2287 to (313.26, 30.6, -154.5) mm, rotated rx -179.9 ry 0 rz -90 deg; joints [36.883, -65.932, 103.318, -128.229, 49.807, 141.585]
  MoveL 2288 to (313.06, 30.52, -156.68) mm, rotated rx -179.9 ry 0 rz -90 deg; joints [36.825, -65.832, 103.178, -128.263, 49.747, 141.583]
  MoveL 2289 to (313.66, 30.44, -158.78) mm, rotated rx -179.9 ry 0 rz -90 deg; joints [36.793, -65.706, 103.002, -128.261, 49.696, 141.551]
  MoveL 2290 to (314.96, 30.37, -160.54) mm, rotated rx -179.9 ry 0 rz -90 deg; joints [36.793, -65.572, 102.812, -128.225, 49.661, 141.494]
  MoveL 2291 to (316.81, 30.29, -161.71) mm, rotated rx -179.9 ry 0 rz -90 deg; joints [36.824, -65.446, 102.633, -128.158, 49.648, 141.42]
  MoveL 2292 to (318.95, 30.21, -162.15) mm, rotated rx -179.9 ry 0 rz -90 deg; joints [36.881, -65.346, 102.491, -128.071, 49.658, 141.339]
  MoveL 2293 to (321.11, 30.14, -161.8) mm, rotated rx -179.9 ry 0 rz -90 deg; joints [36.958, -65.283, 102.402, -127.976, 49.69, 141.264]
  MoveL 2294 to (323, 30.06, -160.7) mm, rotated rx -179.9 ry 0 rz -90 deg; joints [37.044, -65.265, 102.381, -127.885, 49.742, 141.204]
  MoveL 2295 to (324.37, 29.98, -159) mm, rotated rx -179.9 ry 0 rz -90 deg; joints [37.128, -65.295, 102.429, -127.812, 49.806, 141.168]
  MoveL 2296 to (325.05, 29.91, -156.92) mm, rotated rx -179.9 ry 0 rz -90 deg; joints [37.199, -65.369, 102.541, -127.765, 49.874, 141.163]
  MoveL 2297 to (324.94, 29.83, -154.73) mm, rotated rx -179.9 ry 0 rz -90 deg; joints [37.248, -65.476, 102.702, -127.751, 49.938, 141.187]
  MoveL 2298 to (324.06, 29.75, -152.73) mm, rotated rx -179.9 ry 0 rz -90 deg; joints [37.269, -65.602, 102.892, -127.773, 49.99, 141.24]
  MoveL 2299 to (322.53, 29.68, -151.17) mm, rotated rx -179.9 ry 0 rz -90 deg; joints [37.258, -65.73, 103.085, -127.827, 50.023, 141.314]
  MoveL 2300 to (320.54, 29.6, -150.27) mm, rotated rx -179.9 ry 0 rz -90 deg; joints [37.217, -65.844, 103.257, -127.907, 50.033, 141.401]
  MoveL 2301 to (318.36, 29.52, -150.13) mm, rotated rx -179.9 ry 0 rz -90 deg; joints [37.151, -65.927, 103.386, -128.005, 50.02, 141.49]
  MoveL 2302 to (316.27, 29.45, -150.77) mm, rotated rx -179.9 ry 0 rz -90 deg; joints [37.069, -65.969, 103.455, -128.106, 49.986, 141.57]
  MoveL 2303 to (314.55, 29.37, -152.12) mm, rotated rx -179.9 ry 0 rz -90 deg; joints [36.982, -65.964, 103.455, -128.199, 49.935, 141.631]
  MoveL 2304 to (313.42, 29.29, -154) mm, rotated rx -179.9 ry 0 rz -90 deg; joints [36.901, -65.911, 103.387, -128.271, 49.874, 141.667]
  MoveL 2305 to (313.04, 29.22, -156.15) mm, rotated rx -179.9 ry 0 rz -90 deg; joints [36.837, -65.819, 103.26, -128.313, 49.813, 141.672]
  MoveL 2306 to (313.44, 29.14, -158.3) mm, rotated rx -179.9 ry 0 rz -90 deg; joints [36.799, -65.698, 103.09, -128.32, 49.759, 141.647]
  MoveL 2307 to (314.59, 29.06, -160.16) mm, rotated rx -179.9 ry 0 rz -90 deg; joints [36.791, -65.564, 102.901, -128.291, 49.72, 141.595]
  MoveL 2308 to (316.32, 28.99, -161.49) mm, rotated rx -179.9 ry 0 rz -90 deg; joints [36.814, -65.435, 102.718, -128.231, 49.701, 141.524]
  MoveL 2309 to (318.42, 28.91, -162.11) mm, rotated rx -179.9 ry 0 rz -90 deg; joints [36.866, -65.327, 102.564, -128.148, 49.705, 141.444]
  MoveL 2310 to (320.6, 28.83, -161.95) mm, rotated rx -179.9 ry 0 rz -90 deg; joints [36.939, -65.254, 102.461, -128.054, 49.732, 141.366]
  MoveL 2311 to (322.58, 28.76, -161.02) mm, rotated rx -179.9 ry 0 rz -90 deg; joints [37.023, -65.225, 102.423, -127.961, 49.779, 141.302]
  MoveL 2312 to (324.1, 28.68, -159.45) mm, rotated rx -179.9 ry 0 rz -90 deg; joints [37.109, -65.244, 102.454, -127.882, 49.841, 141.26]
  MoveL 2313 to (324.95, 28.6, -157.44) mm, rotated rx -179.9 ry 0 rz -90 deg; joints [37.184, -65.308, 102.552, -127.828, 49.909, 141.247]
  MoveL 2314 to (325.04, 28.53, -155.26) mm, rotated rx -179.9 ry 0 rz -90 deg; joints [37.24, -65.408, 102.703, -127.806, 49.975, 141.264]
  MoveL 2315 to (324.34, 28.45, -153.19) mm, rotated rx -179.9 ry 0 rz -90 deg; joints [37.267, -65.53, 102.888, -127.819, 50.03, 141.31]
  MoveL 2316 to (322.95, 28.37, -151.5) mm, rotated rx -179.9 ry 0 rz -90 deg; joints [37.264, -65.66, 103.082, -127.866, 50.069, 141.38]
  MoveL 2317 to (321.05, 28.3, -150.42) mm, rotated rx -179.9 ry 0 rz -90 deg; joints [37.23, -65.778, 103.262, -127.941, 50.085, 141.465]
  MoveL 2318 to (318.89, 28.22, -150.09) mm, rotated rx -179.9 ry 0 rz -90 deg; joints [37.17, -65.87, 103.403, -128.035, 50.077, 141.554]
  MoveL 2319 to (316.75, 28.14, -150.55) mm, rotated rx -179.9 ry 0 rz -90 deg; joints [37.091, -65.923, 103.488, -128.136, 50.048, 141.637]
  MoveL 2320 to (314.92, 28.06, -151.74) mm, rotated rx -179.9 ry 0 rz -90 deg; joints [37.004, -65.929, 103.505, -128.232, 50, 141.704]
  MoveL 2321 to (313.63, 27.99, -153.51) mm, rotated rx -179.9 ry 0 rz -90 deg; joints [36.92, -65.888, 103.453, -128.31, 49.942, 141.746]
  MoveL 2322 to (313.06, 27.91, -155.62) mm, rotated rx -179.9 ry 0 rz -90 deg; joints [36.851, -65.804, 103.338, -128.361, 49.88, 141.759]
  MoveL 2323 to (313.27, 27.83, -157.79) mm, rotated rx -179.9 ry 0 rz -90 deg; joints [36.806, -65.688, 103.177, -128.376, 49.823, 141.741]
  MoveL 2324 to (314.25, 27.76, -159.75) mm, rotated rx -179.9 ry 0 rz -90 deg; joints [36.791, -65.556, 102.991, -128.356, 49.78, 141.695]
  MoveL 2325 to (315.86, 27.68, -161.23) mm, rotated rx -179.9 ry 0 rz -90 deg; joints [36.807, -65.425, 102.803, -128.303, 49.755, 141.628]
  MoveL 2326 to (317.89, 27.6, -162.03) mm, rotated rx -179.9 ry 0 rz -90 deg; joints [36.852, -65.31, 102.641, -128.225, 49.753, 141.549]
  MoveL 2327 to (320.08, 27.53, -162.06) mm, rotated rx -179.9 ry 0 rz -90 deg; joints [36.92, -65.228, 102.524, -128.132, 49.775, 141.47]
  MoveL 2328 to (322.13, 27.45, -161.31) mm, rotated rx -179.9 ry 0 rz -90 deg; joints [37.003, -65.188, 102.469, -128.037, 49.818, 141.401]
  MoveL 2329 to (323.78, 27.37, -159.88) mm, rotated rx -179.9 ry 0 rz -90 deg; joints [37.09, -65.195, 102.484, -127.954, 49.876, 141.353]
  MoveL 2330 to (324.81, 27.3, -157.95) mm, rotated rx -179.9 ry 0 rz -90 deg; joints [37.168, -65.248, 102.566, -127.893, 49.944, 141.333]
  MoveL 2331 to (325.09, 27.22, -155.79) mm, rotated rx -179.9 ry 0 rz -90 deg; joints [37.229, -65.341, 102.705, -127.863, 50.011, 141.343]
  MoveL 2332 to (324.58, 27.14, -153.66) mm, rotated rx -179.9 ry 0 rz -90 deg; joints [37.264, -65.459, 102.884, -127.867, 50.07, 141.382]
  MoveL 2333 to (323.34, 27.07, -151.86) mm, rotated rx -179.9 ry 0 rz -90 deg; joints [37.269, -65.588, 103.079, -127.906, 50.113, 141.447]
  MoveL 2334 to (321.54, 26.99, -150.62) mm, rotated rx -179.9 ry 0 rz -90 deg; joints [37.242, -65.711, 103.265, -127.975, 50.135, 141.529]
  MoveL 2335 to (319.42, 26.91, -150.1) mm, rotated rx -179.9 ry 0 rz -90 deg; joints [37.187, -65.811, 103.417, -128.065, 50.133, 141.618]
  MoveL 2336 to (317.25, 26.84, -150.37) mm, rotated rx -179.9 ry 0 rz -90 deg; joints [37.112, -65.873, 103.517, -128.166, 50.109, 141.703]
  MoveL 2337 to (315.32, 26.76, -151.39) mm, rotated rx -179.9 ry 0 rz -90 deg; joints [37.026, -65.891, 103.55, -128.264, 50.065, 141.775]
  MoveL 2338 to (313.88, 26.68, -153.04) mm, rotated rx -179.9 ry 0 rz -90 deg; joints [36.94, -65.861, 103.515, -128.348, 50.009, 141.824]
  MoveL 2339 to (313.12, 26.61, -155.09) mm, rotated rx -179.9 ry 0 rz -90 deg; joints [36.867, -65.787, 103.414, -128.406, 49.947, 141.844]
  MoveL 2340 to (313.15, 26.53, -157.27) mm, rotated rx -179.9 ry 0 rz -90 deg; joints [36.815, -65.678, 103.263, -128.43, 49.888, 141.833]
  MoveL 2341 to (313.95, 26.45, -159.31) mm, rotated rx -179.9 ry 0 rz -90 deg; joints [36.792, -65.549, 103.08, -128.419, 49.841, 141.794]
  MoveL 2342 to (315.42, 26.38, -160.92) mm, rotated rx -179.9 ry 0 rz -90 deg; joints [36.801, -65.415, 102.891, -128.373, 49.811, 141.731]
  MoveL 2343 to (317.37, 26.3, -161.91) mm, rotated rx -179.9 ry 0 rz -90 deg; joints [36.839, -65.295, 102.72, -128.3, 49.804, 141.654]
  MoveL 2344 to (319.55, 26.22, -162.13) mm, rotated rx -179.9 ry 0 rz -90 deg; joints [36.903, -65.204, 102.59, -128.21, 49.82, 141.573]
  MoveL 2345 to (321.66, 26.15, -161.56) mm, rotated rx -179.9 ry 0 rz -90 deg; joints [36.983, -65.153, 102.519, -128.114, 49.858, 141.501]
  MoveL 2346 to (323.43, 26.07, -160.28) mm, rotated rx -179.9 ry 0 rz -90 deg; joints [37.07, -65.149, 102.517, -128.027, 49.913, 141.448]
  MoveL 2347 to (324.63, 25.99, -158.45) mm, rotated rx -179.9 ry 0 rz -90 deg; joints [37.151, -65.192, 102.583, -127.96, 49.979, 141.42]
  MoveL 2348 to (325.1, 25.92, -156.32) mm, rotated rx -179.9 ry 0 rz -90 deg; joints [37.217, -65.275, 102.71, -127.921, 50.047, 141.423]
  MoveL 2349 to (324.77, 25.84, -154.16) mm, rotated rx -179.9 ry 0 rz -90 deg; joints [37.259, -65.389, 102.881, -127.917, 50.108, 141.455]
  MoveL 2350 to (323.7, 25.76, -152.25) mm, rotated rx -179.9 ry 0 rz -90 deg; joints [37.271, -65.517, 103.075, -127.948, 50.156, 141.515]
  MoveL 2351 to (322.02, 25.69, -150.86) mm, rotated rx -179.9 ry 0 rz -90 deg; joints [37.252, -65.642, 103.265, -128.01, 50.183, 141.593]
  MoveL 2352 to (319.95, 25.61, -150.15) mm, rotated rx -179.9 ry 0 rz -90 deg; joints [37.203, -65.749, 103.427, -128.096, 50.188, 141.681]
  MoveL 2353 to (317.76, 25.53, -150.23) mm, rotated rx -179.9 ry 0 rz -90 deg; joints [37.132, -65.822, 103.541, -128.195, 50.169, 141.769]
  MoveL 2354 to (315.75, 25.45, -151.08) mm, rotated rx -179.9 ry 0 rz -90 deg; joints [37.047, -65.851, 103.592, -128.296, 50.13, 141.845]
  MoveL 2355 to (314.17, 25.38, -152.59) mm, rotated rx -179.9 ry 0 rz -90 deg; joints [36.961, -65.832, 103.573, -128.384, 50.076, 141.9]
  MoveL 2356 to (313.24, 25.3, -154.57) mm, rotated rx -179.9 ry 0 rz -90 deg; joints [36.884, -65.768, 103.487, -128.449, 50.014, 141.927]
  MoveL 2357 to (313.07, 25.22, -156.75) mm, rotated rx -179.9 ry 0 rz -90 deg; joints [36.826, -65.666, 103.346, -128.482, 49.954, 141.924]
  MoveL 2358 to (313.69, 25.15, -158.84) mm, rotated rx -179.9 ry 0 rz -90 deg; joints [36.796, -65.541, 103.169, -128.479, 49.903, 141.891]
  MoveL 2359 to (315.01, 25.07, -160.58) mm, rotated rx -179.9 ry 0 rz -90 deg; joints [36.796, -65.407, 102.979, -128.442, 49.869, 141.833]
  MoveL 2360 to (316.87, 24.99, -161.74) mm, rotated rx -179.9 ry 0 rz -90 deg; joints [36.828, -65.282, 102.801, -128.374, 49.855, 141.758]
  MoveL 2361 to (319.02, 24.92, -162.15) mm, rotated rx -179.9 ry 0 rz -90 deg; joints [36.886, -65.183, 102.66, -128.287, 49.866, 141.678]
  MoveL 2362 to (321.17, 24.84, -161.77) mm, rotated rx -179.9 ry 0 rz -90 deg; joints [36.963, -65.121, 102.573, -128.192, 49.898, 141.602]
  MoveL 2363 to (323.05, 24.76, -160.65) mm, rotated rx -179.9 ry 0 rz -90 deg; joints [37.049, -65.105, 102.554, -128.101, 49.95, 141.544]
  MoveL 2364 to (324.4, 24.69, -158.94) mm, rotated rx -179.9 ry 0 rz -90 deg; joints [37.133, -65.137, 102.604, -128.028, 50.014, 141.509]
  MoveL 2365 to (325.06, 24.61, -156.85) mm, rotated rx -179.9 ry 0 rz -90 deg; joints [37.204, -65.211, 102.717, -127.982, 50.082, 141.504]
  MoveL 2366 to (324.92, 24.53, -154.67) mm, rotated rx -179.9 ry 0 rz -90 deg; joints [37.252, -65.319, 102.88, -127.969, 50.146, 141.53]
  MoveL 2367 to (324.02, 24.46, -152.68) mm, rotated rx -179.9 ry 0 rz -90 deg; joints [37.272, -65.445, 103.07, -127.991, 50.198, 141.583]
  MoveL 2368 to (322.47, 24.38, -151.14) mm, rotated rx -179.9 ry 0 rz -90 deg; joints [37.26, -65.572, 103.263, -128.046, 50.231, 141.658]
  MoveL 2369 to (320.47, 24.3, -150.25) mm, rotated rx -179.9 ry 0 rz -90 deg; joints [37.218, -65.685, 103.434, -128.127, 50.241, 141.745]
  MoveL 2370 to (318.29, 24.23, -150.14) mm, rotated rx -179.9 ry 0 rz -90 deg; joints [37.152, -65.767, 103.562, -128.225, 50.228, 141.833]
  MoveL 2371 to (316.21, 24.15, -150.81) mm, rotated rx -179.9 ry 0 rz -90 deg; joints [37.069, -65.807, 103.629, -128.326, 50.193, 141.913]
  MoveL 2372 to (314.5, 24.07, -152.17) mm, rotated rx -179.9 ry 0 rz -90 deg; joints [36.982, -65.8, 103.627, -128.418, 50.142, 141.974]
  MoveL 2373 to (313.4, 24, -154.06) mm, rotated rx -179.9 ry 0 rz -90 deg; joints [36.902, -65.747, 103.556, -128.49, 50.082, 142.008]
  MoveL 2374 to (313.04, 23.92, -156.22) mm, rotated rx -179.9 ry 0 rz -90 deg; joints [36.838, -65.653, 103.427, -128.531, 50.021, 142.012]
  MoveL 2375 to (313.47, 23.84, -158.36) mm, rotated rx -179.9 ry 0 rz -90 deg; joints [36.801, -65.532, 103.257, -128.538, 49.967, 141.986]
  MoveL 2376 to (314.63, 23.77, -160.21) mm, rotated rx -179.9 ry 0 rz -90 deg; joints [36.794, -65.398, 103.067, -128.508, 49.928, 141.934]
  MoveL 2377 to (316.38, 23.69, -161.52) mm, rotated rx -179.9 ry 0 rz -90 deg; joints [36.818, -65.27, 102.884, -128.447, 49.909, 141.862]
  MoveL 2378 to (318.48, 23.61, -162.12) mm, rotated rx -179.9 ry 0 rz -90 deg; joints [36.87, -65.163, 102.732, -128.363, 49.913, 141.782]
  MoveL 2379 to (320.66, 23.54, -161.94) mm, rotated rx -179.9 ry 0 rz -90 deg; joints [36.944, -65.092, 102.631, -128.269, 49.94, 141.704]
  MoveL 2380 to (322.63, 23.46, -160.99) mm, rotated rx -179.9 ry 0 rz -90 deg; joints [37.029, -65.064, 102.595, -128.176, 49.988, 141.641]
  MoveL 2381 to (324.13, 23.38, -159.4) mm, rotated rx -179.9 ry 0 rz -90 deg; joints [37.114, -65.085, 102.628, -128.098, 50.049, 141.6]
  MoveL 2382 to (324.97, 23.31, -157.38) mm, rotated rx -179.9 ry 0 rz -90 deg; joints [37.189, -65.149, 102.727, -128.044, 50.117, 141.588]
  MoveL 2383 to (325.03, 23.23, -155.19) mm, rotated rx -179.9 ry 0 rz -90 deg; joints [37.244, -65.25, 102.88, -128.023, 50.183, 141.606]
  MoveL 2384 to (324.31, 23.15, -153.13) mm, rotated rx -179.9 ry 0 rz -90 deg; joints [37.271, -65.373, 103.065, -128.037, 50.238, 141.653]
  MoveL 2385 to (322.9, 23.08, -151.46) mm, rotated rx -179.9 ry 0 rz -90 deg; joints [37.266, -65.502, 103.26, -128.084, 50.276, 141.723]
  MoveL 2386 to (320.98, 23, -150.4) mm, rotated rx -179.9 ry 0 rz -90 deg; joints [37.231, -65.619, 103.439, -128.16, 50.293, 141.808]
  MoveL 2387 to (318.82, 22.92, -150.09) mm, rotated rx -179.9 ry 0 rz -90 deg; joints [37.17, -65.71, 103.579, -128.254, 50.285, 141.897]
  MoveL 2388 to (316.69, 22.84, -150.57) mm, rotated rx -179.9 ry 0 rz -90 deg; joints [37.091, -65.761, 103.661, -128.356, 50.255, 141.98]
  MoveL 2389 to (314.87, 22.77, -151.79) mm, rotated rx -179.9 ry 0 rz -90 deg; joints [37.004, -65.765, 103.676, -128.452, 50.208, 142.046]
  MoveL 2390 to (313.6, 22.69, -153.57) mm, rotated rx -179.9 ry 0 rz -90 deg; joints [36.92, -65.723, 103.622, -128.529, 50.149, 142.087]
  MoveL 2391 to (313.05, 22.61, -155.68) mm, rotated rx -179.9 ry 0 rz -90 deg; joints [36.852, -65.638, 103.506, -128.578, 50.088, 142.099]
  MoveL 2392 to (313.29, 22.54, -157.86) mm, rotated rx -179.9 ry 0 rz -90 deg; joints [36.808, -65.522, 103.343, -128.593, 50.031, 142.08]
  MoveL 2393 to (314.29, 22.46, -159.8) mm, rotated rx -179.9 ry 0 rz -90 deg; joints [36.793, -65.39, 103.156, -128.572, 49.988, 142.033]
  MoveL 2394 to (315.92, 22.38, -161.26) mm, rotated rx -179.9 ry 0 rz -90 deg; joints [36.81, -65.259, 102.969, -128.518, 49.963, 141.965]
  MoveL 2395 to (317.96, 22.31, -162.05) mm, rotated rx -179.9 ry 0 rz -90 deg; joints [36.856, -65.146, 102.808, -128.439, 49.962, 141.886]
  MoveL 2396 to (320.14, 22.23, -162.05) mm, rotated rx -179.9 ry 0 rz -90 deg; joints [36.925, -65.065, 102.693, -128.346, 49.984, 141.807]
  MoveL 2397 to (322.19, 22.15, -161.28) mm, rotated rx -179.9 ry 0 rz -90 deg; joints [37.008, -65.026, 102.64, -128.252, 50.026, 141.739]
  MoveL 2398 to (323.82, 22.08, -159.83) mm, rotated rx -179.9 ry 0 rz -90 deg; joints [37.095, -65.035, 102.656, -128.169, 50.085, 141.692]
  MoveL 2399 to (324.83, 22, -157.89) mm, rotated rx -179.9 ry 0 rz -90 deg; joints [37.173, -65.089, 102.741, -128.109, 50.152, 141.672]
  MoveL 2400 to (325.09, 21.92, -155.72) mm, rotated rx -179.9 ry 0 rz -90 deg; joints [37.233, -65.182, 102.882, -128.079, 50.219, 141.684]
  MoveL 2401 to (324.55, 21.85, -153.6) mm, rotated rx -179.9 ry 0 rz -90 deg; joints [37.267, -65.301, 103.061, -128.084, 50.278, 141.724]
  MoveL 2402 to (323.29, 21.77, -151.81) mm, rotated rx -179.9 ry 0 rz -90 deg; joints [37.271, -65.43, 103.256, -128.124, 50.321, 141.79]
  MoveL 2403 to (321.48, 21.69, -150.59) mm, rotated rx -179.9 ry 0 rz -90 deg; joints [37.243, -65.552, 103.441, -128.193, 50.343, 141.872]
  MoveL 2404 to (319.35, 21.62, -150.09) mm, rotated rx -179.9 ry 0 rz -90 deg; joints [37.188, -65.65, 103.592, -128.284, 50.341, 141.961]
  MoveL 2405 to (317.19, 21.54, -150.39) mm, rotated rx -179.9 ry 0 rz -90 deg; joints [37.112, -65.711, 103.69, -128.385, 50.317, 142.046]
  MoveL 2406 to (315.27, 21.46, -151.43) mm, rotated rx -179.9 ry 0 rz -90 deg; joints [37.026, -65.728, 103.722, -128.483, 50.273, 142.117]
  MoveL 2407 to (313.85, 21.39, -153.1) mm, rotated rx -179.9 ry 0 rz -90 deg; joints [36.94, -65.696, 103.684, -128.566, 50.217, 142.165]
  MoveL 2408 to (313.11, 21.31, -155.15) mm, rotated rx -179.9 ry 0 rz -90 deg; joints [36.868, -65.621, 103.581, -128.623, 50.155, 142.184]
  MoveL 2409 to (313.16, 21.23, -157.34) mm, rotated rx -179.9 ry 0 rz -90 deg; joints [36.817, -65.512, 103.428, -128.647, 50.096, 142.172]
  MoveL 2410 to (313.98, 21.16, -159.37) mm, rotated rx -179.9 ry 0 rz -90 deg; joints [36.795, -65.382, 103.245, -128.635, 50.049, 142.131]
  MoveL 2411 to (315.48, 21.08, -160.96) mm, rotated rx -179.9 ry 0 rz -90 deg; joints [36.804, -65.249, 103.056, -128.588, 50.02, 142.068]
  MoveL 2412 to (317.44, 21, -161.93) mm, rotated rx -179.9 ry 0 rz -90 deg; joints [36.843, -65.13, 102.886, -128.514, 50.012, 141.99]
  MoveL 2413 to (319.62, 20.93, -162.13) mm, rotated rx -179.9 ry 0 rz -90 deg; joints [36.908, -65.04, 102.758, -128.423, 50.028, 141.91]
  MoveL 2414 to (321.72, 20.85, -161.54) mm, rotated rx -179.9 ry 0 rz -90 deg; joints [36.988, -64.991, 102.689, -128.328, 50.066, 141.839]
  MoveL 2415 to (323.48, 20.77, -160.23) mm, rotated rx -179.9 ry 0 rz -90 deg; joints [37.075, -64.988, 102.688, -128.241, 50.122, 141.786]
  MoveL 2416 to (324.66, 20.7, -158.39) mm, rotated rx -179.9 ry 0 rz -90 deg; joints [37.156, -65.032, 102.757, -128.174, 50.187, 141.759]
  MoveL 2417 to (325.1, 20.62, -156.25) mm, rotated rx -179.9 ry 0 rz -90 deg; joints [37.222, -65.116, 102.885, -128.137, 50.255, 141.763]
  MoveL 2418 to (324.75, 20.54, -154.09) mm, rotated rx -179.9 ry 0 rz -90 deg; joints [37.263, -65.23, 103.058, -128.133, 50.317, 141.796]
  MoveL 2419 to (323.66, 20.47, -152.2) mm, rotated rx -179.9 ry 0 rz -90 deg; joints [37.274, -65.358, 103.251, -128.165, 50.364, 141.856]
  MoveL 2420 to (321.96, 20.39, -150.82) mm, rotated rx -179.9 ry 0 rz -90 deg; joints [37.253, -65.483, 103.441, -128.227, 50.392, 141.935]
  MoveL 2421 to (319.88, 20.31, -150.14) mm, rotated rx -179.9 ry 0 rz -90 deg; joints [37.204, -65.588, 103.602, -128.314, 50.396, 142.024]
  MoveL 2422 to (317.7, 20.23, -150.24) mm, rotated rx -179.9 ry 0 rz -90 deg; joints [37.132, -65.659, 103.714, -128.414, 50.377, 142.111]
  MoveL 2423 to (315.7, 20.16, -151.12) mm, rotated rx -179.9 ry 0 rz -90 deg; joints [37.047, -65.687, 103.763, -128.514, 50.338, 142.186]
  MoveL 2424 to (314.13, 20.08, -152.65) mm, rotated rx -179.9 ry 0 rz -90 deg; joints [36.961, -65.667, 103.742, -128.602, 50.284, 142.24]
  MoveL 2425 to (313.22, 20, -154.63) mm, rotated rx -179.9 ry 0 rz -90 deg; joints [36.884, -65.602, 103.654, -128.666, 50.222, 142.266]
  MoveL 2426 to (313.08, 19.93, -156.81) mm, rotated rx -179.9 ry 0 rz -90 deg; joints [36.827, -65.499, 103.511, -128.698, 50.162, 142.262]
  MoveL 2427 to (313.72, 19.85, -158.9) mm, rotated rx -179.9 ry 0 rz -90 deg; joints [36.798, -65.373, 103.333, -128.695, 50.112, 142.228]
  MoveL 2428 to (315.06, 19.77, -160.63) mm, rotated rx -179.9 ry 0 rz -90 deg; joints [36.799, -65.24, 103.143, -128.656, 50.077, 142.169]
  MoveL 2429 to (316.93, 19.7, -161.76) mm, rotated rx -179.9 ry 0 rz -90 deg; joints [36.832, -65.116, 102.966, -128.588, 50.064, 142.094]
  MoveL 2430 to (319.08, 19.62, -162.15) mm, rotated rx -179.9 ry 0 rz -90 deg; joints [36.891, -65.018, 102.826, -128.5, 50.074, 142.014]
  MoveL 2431 to (321.23, 19.54, -161.75) mm, rotated rx -179.9 ry 0 rz -90 deg; joints [36.968, -64.958, 102.742, -128.405, 50.107, 141.939]
  MoveL 2432 to (323.1, 19.47, -160.61) mm, rotated rx -179.9 ry 0 rz -90 deg; joints [37.055, -64.944, 102.724, -128.315, 50.159, 141.881]
  MoveL 2433 to (324.43, 19.39, -158.88) mm, rotated rx -179.9 ry 0 rz -90 deg; joints [37.138, -64.976, 102.777, -128.242, 50.223, 141.847]
  MoveL 2434 to (325.06, 19.31, -156.78) mm, rotated rx -179.9 ry 0 rz -90 deg; joints [37.208, -65.052, 102.892, -128.196, 50.291, 141.844]
  MoveL 2435 to (324.91, 19.24, -154.6) mm, rotated rx -179.9 ry 0 rz -90 deg; joints [37.256, -65.16, 103.055, -128.184, 50.355, 141.87]
  MoveL 2436 to (323.98, 19.16, -152.62) mm, rotated rx -179.9 ry 0 rz -90 deg; joints [37.275, -65.286, 103.246, -128.207, 50.406, 141.924]
  MoveL 2437 to (322.42, 19.08, -151.1) mm, rotated rx -179.9 ry 0 rz -90 deg; joints [37.262, -65.413, 103.439, -128.263, 50.439, 142]
  MoveL 2438 to (320.41, 19.01, -150.24) mm, rotated rx -179.9 ry 0 rz -90 deg; joints [37.219, -65.524, 103.609, -128.345, 50.449, 142.087]
  MoveL 2439 to (318.22, 18.93, -150.14) mm, rotated rx -179.9 ry 0 rz -90 deg; joints [37.152, -65.605, 103.735, -128.443, 50.436, 142.175]
  MoveL 2440 to (316.15, 18.85, -150.84) mm, rotated rx -179.9 ry 0 rz -90 deg; joints [37.069, -65.643, 103.8, -128.544, 50.401, 142.254]
  MoveL 2441 to (314.46, 18.78, -152.23) mm, rotated rx -179.9 ry 0 rz -90 deg; joints [36.982, -65.635, 103.795, -128.636, 50.35, 142.314]
  MoveL 2442 to (313.37, 18.7, -154.12) mm, rotated rx -179.9 ry 0 rz -90 deg; joints [36.902, -65.58, 103.723, -128.707, 50.29, 142.347]
  MoveL 2443 to (313.04, 18.62, -156.28) mm, rotated rx -179.9 ry 0 rz -90 deg; joints [36.839, -65.486, 103.592, -128.747, 50.229, 142.35]
  MoveL 2444 to (313.49, 18.55, -158.42) mm, rotated rx -179.9 ry 0 rz -90 deg; joints [36.803, -65.364, 103.421, -128.752, 50.175, 142.323]
  MoveL 2445 to (314.68, 18.47, -160.26) mm, rotated rx -179.9 ry 0 rz -90 deg; joints [36.797, -65.231, 103.231, -128.722, 50.136, 142.269]
  MoveL 2446 to (316.44, 18.39, -161.55) mm, rotated rx -179.9 ry 0 rz -90 deg; joints [36.822, -65.103, 103.049, -128.66, 50.117, 142.198]
  MoveL 2447 to (318.55, 18.32, -162.13) mm, rotated rx -179.9 ry 0 rz -90 deg; joints [36.875, -64.998, 102.898, -128.576, 50.122, 142.117]
  MoveL 2448 to (320.73, 18.24, -161.92) mm, rotated rx -179.9 ry 0 rz -90 deg; joints [36.949, -64.928, 102.799, -128.481, 50.149, 142.04]
  MoveL 2449 to (322.69, 18.16, -160.95) mm, rotated rx -179.9 ry 0 rz -90 deg; joints [37.034, -64.902, 102.764, -128.389, 50.197, 141.977]
  MoveL 2450 to (324.17, 18.09, -159.34) mm, rotated rx -179.9 ry 0 rz -90 deg; joints [37.119, -64.923, 102.8, -128.311, 50.258, 141.937]
  MoveL 2451 to (324.98, 18.01, -157.31) mm, rotated rx -179.9 ry 0 rz -90 deg; joints [37.194, -64.989, 102.901, -128.258, 50.326, 141.926]
  MoveL 2452 to (325.02, 17.93, -155.12) mm, rotated rx -179.9 ry 0 rz -90 deg; joints [37.248, -65.09, 103.055, -128.237, 50.392, 141.945]
  MoveL 2453 to (324.27, 17.85, -153.07) mm, rotated rx -179.9 ry 0 rz -90 deg; joints [37.274, -65.213, 103.241, -128.252, 50.447, 141.993]
  MoveL 2454 to (322.84, 17.78, -151.41) mm, rotated rx -179.9 ry 0 rz -90 deg; joints [37.268, -65.342, 103.436, -128.3, 50.485, 142.064]
  MoveL 2455 to (320.92, 17.7, -150.38) mm, rotated rx -179.9 ry 0 rz -90 deg; joints [37.233, -65.458, 103.613, -128.376, 50.501, 142.149]
  MoveL 2456 to (318.75, 17.62, -150.09) mm, rotated rx -179.9 ry 0 rz -90 deg; joints [37.171, -65.547, 103.752, -128.471, 50.493, 142.238]
  MoveL 2457 to (316.63, 17.55, -150.6) mm, rotated rx -179.9 ry 0 rz -90 deg; joints [37.091, -65.597, 103.832, -128.573, 50.464, 142.32]
  MoveL 2458 to (314.82, 17.47, -151.83) mm, rotated rx -179.9 ry 0 rz -90 deg; joints [37.004, -65.6, 103.845, -128.668, 50.416, 142.386]
  MoveL 2459 to (313.57, 17.39, -153.63) mm, rotated rx -179.9 ry 0 rz -90 deg; joints [36.921, -65.556, 103.789, -128.745, 50.358, 142.426]
  MoveL 2460 to (313.05, 17.32, -155.75) mm, rotated rx -179.9 ry 0 rz -90 deg; joints [36.853, -65.47, 103.671, -128.794, 50.296, 142.436]
  MoveL 2461 to (313.31, 17.24, -157.92) mm, rotated rx -179.9 ry 0 rz -90 deg; joints [36.81, -65.354, 103.507, -128.808, 50.24, 142.416]
  MoveL 2462 to (314.33, 17.16, -159.85) mm, rotated rx -179.9 ry 0 rz -90 deg; joints [36.796, -65.222, 103.32, -128.786, 50.196, 142.369]
  MoveL 2463 to (315.97, 17.09, -161.3) mm, rotated rx -179.9 ry 0 rz -90 deg; joints [36.814, -65.092, 103.133, -128.731, 50.172, 142.3]
  MoveL 2464 to (318.02, 17.01, -162.06) mm, rotated rx -179.9 ry 0 rz -90 deg; joints [36.861, -64.98, 102.973, -128.652, 50.171, 142.221]
  MoveL 2465 to (320.21, 16.93, -162.04) mm, rotated rx -179.9 ry 0 rz -90 deg; joints [36.93, -64.9, 102.859, -128.558, 50.193, 142.142]
  MoveL 2466 to (322.25, 16.86, -161.25) mm, rotated rx -179.9 ry 0 rz -90 deg; joints [37.014, -64.863, 102.808, -128.464, 50.236, 142.075]
  MoveL 2467 to (323.86, 16.78, -159.78) mm, rotated rx -179.9 ry 0 rz -90 deg; joints [37.1, -64.873, 102.827, -128.381, 50.294, 142.029]
  MoveL 2468 to (324.85, 16.7, -157.83) mm, rotated rx -179.9 ry 0 rz -90 deg; joints [37.178, -64.929, 102.913, -128.321, 50.361, 142.01]
  MoveL 2469 to (325.08, 16.63, -155.65) mm, rotated rx -179.9 ry 0 rz -90 deg; joints [37.237, -65.022, 103.056, -128.292, 50.429, 142.022]
  MoveL 2470 to (324.52, 16.55, -153.54) mm, rotated rx -179.9 ry 0 rz -90 deg; joints [37.271, -65.141, 103.236, -128.298, 50.487, 142.064]
  MoveL 2471 to (323.25, 16.47, -151.76) mm, rotated rx -179.9 ry 0 rz -90 deg; joints [37.273, -65.27, 103.431, -128.339, 50.53, 142.13]
  MoveL 2472 to (321.42, 16.4, -150.56) mm, rotated rx -179.9 ry 0 rz -90 deg; joints [37.245, -65.391, 103.615, -128.409, 50.552, 142.212]
  MoveL 2473 to (319.29, 16.32, -150.09) mm, rotated rx -179.9 ry 0 rz -90 deg; joints [37.188, -65.488, 103.765, -128.5, 50.55, 142.301]
  MoveL 2474 to (317.12, 16.24, -150.41) mm, rotated rx -179.9 ry 0 rz -90 deg; joints [37.112, -65.548, 103.861, -128.602, 50.525, 142.386]
  MoveL 2475 to (315.22, 16.17, -151.48) mm, rotated rx -179.9 ry 0 rz -90 deg; joints [37.026, -65.562, 103.89, -128.7, 50.482, 142.456]
  MoveL 2476 to (313.81, 16.09, -153.15) mm, rotated rx -179.9 ry 0 rz -90 deg; joints [36.941, -65.529, 103.85, -128.782, 50.425, 142.503]
  MoveL 2477 to (313.1, 16.01, -155.22) mm, rotated rx -179.9 ry 0 rz -90 deg; joints [36.868, -65.453, 103.746, -128.838, 50.363, 142.521]
  MoveL 2478 to (313.17, 15.94, -157.41) mm, rotated rx -179.9 ry 0 rz -90 deg; joints [36.818, -65.343, 103.592, -128.861, 50.305, 142.508]
  MoveL 2479 to (314.02, 15.86, -159.42) mm, rotated rx -179.9 ry 0 rz -90 deg; joints [36.797, -65.214, 103.408, -128.848, 50.258, 142.466]
  MoveL 2480 to (315.53, 15.78, -161) mm, rotated rx -179.9 ry 0 rz -90 deg; joints [36.807, -65.081, 103.219, -128.8, 50.229, 142.402]
  MoveL 2481 to (317.5, 15.71, -161.94) mm, rotated rx -179.9 ry 0 rz -90 deg; joints [36.848, -64.963, 103.05, -128.726, 50.221, 142.325]
  MoveL 2482 to (319.68, 15.63, -162.12) mm, rotated rx -179.9 ry 0 rz -90 deg; joints [36.913, -64.875, 102.923, -128.635, 50.238, 142.245]
  MoveL 2483 to (321.78, 15.55, -161.51) mm, rotated rx -179.9 ry 0 rz -90 deg; joints [36.994, -64.827, 102.856, -128.539, 50.276, 142.173]
  MoveL 2484 to (323.52, 15.48, -160.18) mm, rotated rx -179.9 ry 0 rz -90 deg; joints [37.08, -64.825, 102.858, -128.453, 50.331, 142.121]
  MoveL 2485 to (324.68, 15.4, -158.33) mm, rotated rx -179.9 ry 0 rz -90 deg; joints [37.161, -64.87, 102.928, -128.387, 50.397, 142.096]
  MoveL 2486 to (325.1, 15.32, -156.18) mm, rotated rx -179.9 ry 0 rz -90 deg; joints [37.226, -64.955, 103.059, -128.35, 50.465, 142.101]
  MoveL 2487 to (324.73, 15.24, -154.03) mm, rotated rx -179.9 ry 0 rz -90 deg; joints [37.266, -65.07, 103.232, -128.347, 50.526, 142.135]
  MoveL 2488 to (323.61, 15.17, -152.15) mm, rotated rx -179.9 ry 0 rz -90 deg; joints [37.276, -65.197, 103.426, -128.379, 50.573, 142.196]
  MoveL 2489 to (321.9, 15.09, -150.79) mm, rotated rx -179.9 ry 0 rz -90 deg; joints [37.255, -65.321, 103.615, -128.443, 50.601, 142.275]
  MoveL 2490 to (319.82, 15.01, -150.13) mm, rotated rx -179.9 ry 0 rz -90 deg; joints [37.205, -65.426, 103.775, -128.53, 50.605, 142.364]
  MoveL 2491 to (317.63, 14.94, -150.26) mm, rotated rx -179.9 ry 0 rz -90 deg; joints [37.132, -65.495, 103.885, -128.63, 50.586, 142.45]
  MoveL 2492 to (315.64, 14.86, -151.15) mm, rotated rx -179.9 ry 0 rz -90 deg; joints [37.047, -65.521, 103.932, -128.73, 50.546, 142.525]
  MoveL 2493 to (314.1, 14.78, -152.7) mm, rotated rx -179.9 ry 0 rz -90 deg; joints [36.961, -65.5, 103.908, -128.817, 50.492, 142.578]
  MoveL 2494 to (313.2, 14.71, -154.7) mm, rotated rx -179.9 ry 0 rz -90 deg; joints [36.885, -65.434, 103.819, -128.881, 50.431, 142.603]
  MoveL 2495 to (313.08, 14.63, -156.88) mm, rotated rx -179.9 ry 0 rz -90 deg; joints [36.829, -65.331, 103.675, -128.912, 50.371, 142.598]
  MoveL 2496 to (313.75, 14.55, -158.96) mm, rotated rx -179.9 ry 0 rz -90 deg; joints [36.8, -65.204, 103.496, -128.907, 50.321, 142.562]
  MoveL 2497 to (315.11, 14.48, -160.67) mm, rotated rx -179.9 ry 0 rz -90 deg; joints [36.803, -65.071, 103.306, -128.868, 50.286, 142.503]
  MoveL 2498 to (317, 14.4, -161.78) mm, rotated rx -179.9 ry 0 rz -90 deg; joints [36.836, -64.948, 103.129, -128.799, 50.273, 142.428]
  MoveL 2499 to (319.15, 14.32, -162.15) mm, rotated rx -179.9 ry 0 rz -90 deg; joints [36.896, -64.852, 102.991, -128.711, 50.284, 142.347]
  MoveL 2500 to (321.3, 14.25, -161.72) mm, rotated rx -179.9 ry 0 rz -90 deg; joints [36.974, -64.793, 102.908, -128.615, 50.317, 142.273]
  MoveL 2501 to (323.15, 14.17, -160.56) mm, rotated rx -179.9 ry 0 rz -90 deg; joints [37.06, -64.78, 102.893, -128.525, 50.368, 142.216]
  MoveL 2502 to (324.46, 14.09, -158.82) mm, rotated rx -179.9 ry 0 rz -90 deg; joints [37.143, -64.814, 102.947, -128.453, 50.432, 142.183]
  MoveL 2503 to (325.07, 14.02, -156.72) mm, rotated rx -179.9 ry 0 rz -90 deg; joints [37.213, -64.89, 103.064, -128.408, 50.5, 142.18]
  MoveL 2504 to (324.89, 13.94, -154.54) mm, rotated rx -179.9 ry 0 rz -90 deg; joints [37.26, -64.999, 103.229, -128.397, 50.564, 142.208]
  MoveL 2505 to (323.94, 13.86, -152.57) mm, rotated rx -179.9 ry 0 rz -90 deg; joints [37.277, -65.125, 103.42, -128.421, 50.616, 142.263]
  MoveL 2506 to (322.36, 13.79, -151.06) mm, rotated rx -179.9 ry 0 rz -90 deg; joints [37.264, -65.251, 103.612, -128.478, 50.648, 142.339]
  MoveL 2507 to (320.34, 13.71, -150.22) mm, rotated rx -179.9 ry 0 rz -90 deg; joints [37.22, -65.361, 103.782, -128.56, 50.658, 142.426]
  MoveL 2508 to (318.16, 13.63, -150.15) mm, rotated rx -179.9 ry 0 rz -90 deg; joints [37.152, -65.44, 103.906, -128.658, 50.645, 142.514]
  MoveL 2509 to (316.09, 13.56, -150.87) mm, rotated rx -179.9 ry 0 rz -90 deg; joints [37.069, -65.478, 103.968, -128.759, 50.61, 142.592]
  MoveL 2510 to (314.42, 13.48, -152.28) mm, rotated rx -179.9 ry 0 rz -90 deg; joints [36.982, -65.468, 103.962, -128.851, 50.559, 142.651]
  MoveL 2511 to (313.35, 13.4, -154.19) mm, rotated rx -179.9 ry 0 rz -90 deg; joints [36.902, -65.412, 103.888, -128.921, 50.499, 142.683]
  MoveL 2512 to (313.04, 13.33, -156.35) mm, rotated rx -179.9 ry 0 rz -90 deg; joints [36.841, -65.317, 103.755, -128.961, 50.438, 142.685]
  MoveL 2513 to (313.52, 13.25, -158.48) mm, rotated rx -179.9 ry 0 rz -90 deg; joints [36.805, -65.195, 103.583, -128.965, 50.384, 142.657]
  MoveL 2514 to (314.73, 13.17, -160.31) mm, rotated rx -179.9 ry 0 rz -90 deg; joints [36.8, -65.062, 103.393, -128.933, 50.346, 142.603]
  MoveL 2515 to (316.5, 13.1, -161.58) mm, rotated rx -179.9 ry 0 rz -90 deg; joints [36.826, -64.935, 103.211, -128.871, 50.327, 142.531]
  MoveL 2516 to (318.62, 13.02, -162.13) mm, rotated rx -179.9 ry 0 rz -90 deg; joints [36.88, -64.831, 103.061, -128.786, 50.332, 142.45]
  MoveL 2517 to (320.79, 12.94, -161.9) mm, rotated rx -179.9 ry 0 rz -90 deg; joints [36.954, -64.762, 102.964, -128.691, 50.359, 142.374]
  MoveL 2518 to (322.74, 12.87, -160.9) mm, rotated rx -179.9 ry 0 rz -90 deg; joints [37.039, -64.738, 102.932, -128.599, 50.407, 142.311]
  MoveL 2519 to (324.2, 12.79, -159.28) mm, rotated rx -179.9 ry 0 rz -90 deg; joints [37.125, -64.76, 102.969, -128.521, 50.468, 142.272]
  MoveL 2520 to (324.99, 12.71, -157.24) mm, rotated rx -179.9 ry 0 rz -90 deg; joints [37.198, -64.827, 103.072, -128.469, 50.536, 142.262]
  MoveL 2521 to (325.01, 12.63, -155.06) mm, rotated rx -179.9 ry 0 rz -90 deg; joints [37.251, -64.929, 103.227, -128.449, 50.602, 142.283]
  MoveL 2522 to (324.24, 12.56, -153.01) mm, rotated rx -179.9 ry 0 rz -90 deg; joints [37.277, -65.052, 103.414, -128.465, 50.657, 142.331]
  MoveL 2523 to (322.79, 12.48, -151.37) mm, rotated rx -179.9 ry 0 rz -90 deg; joints [37.27, -65.18, 103.609, -128.514, 50.695, 142.403]
  MoveL 2524 to (320.86, 12.4, -150.36) mm, rotated rx -179.9 ry 0 rz -90 deg; joints [37.234, -65.295, 103.786, -128.591, 50.71, 142.488]
  MoveL 2525 to (318.69, 12.33, -150.1) mm, rotated rx -179.9 ry 0 rz -90 deg; joints [37.171, -65.383, 103.922, -128.686, 50.703, 142.577]
  MoveL 2526 to (316.57, 12.25, -150.63) mm, rotated rx -179.9 ry 0 rz -90 deg; joints [37.091, -65.431, 104.001, -128.788, 50.673, 142.658]
  MoveL 2527 to (314.77, 12.17, -151.88) mm, rotated rx -179.9 ry 0 rz -90 deg; joints [37.004, -65.433, 104.012, -128.883, 50.625, 142.723]
  MoveL 2528 to (313.55, 12.1, -153.69) mm, rotated rx -179.9 ry 0 rz -90 deg; joints [36.921, -65.388, 103.953, -128.959, 50.567, 142.762]
  MoveL 2529 to (313.04, 12.02, -155.82) mm, rotated rx -179.9 ry 0 rz -90 deg; joints [36.854, -65.301, 103.833, -129.007, 50.505, 142.771]
  MoveL 2530 to (313.33, 11.94, -157.98) mm, rotated rx -179.9 ry 0 rz -90 deg; joints [36.812, -65.184, 103.669, -129.02, 50.449, 142.75]
  MoveL 2531 to (314.37, 11.87, -159.91) mm, rotated rx -179.9 ry 0 rz -90 deg; joints [36.799, -65.053, 103.481, -128.997, 50.406, 142.702]
  MoveL 2532 to (316.03, 11.79, -161.33) mm, rotated rx -179.9 ry 0 rz -90 deg; joints [36.818, -64.923, 103.295, -128.941, 50.382, 142.633]
  MoveL 2533 to (318.09, 11.71, -162.07) mm, rotated rx -179.9 ry 0 rz -90 deg; joints [36.865, -64.812, 103.135, -128.861, 50.381, 142.553]
  MoveL 2534 to (320.28, 11.64, -162.03) mm, rotated rx -179.9 ry 0 rz -90 deg; joints [36.935, -64.733, 103.023, -128.768, 50.403, 142.475]
  MoveL 2535 to (322.3, 11.56, -161.21) mm, rotated rx -179.9 ry 0 rz -90 deg; joints [37.019, -64.698, 102.975, -128.673, 50.446, 142.408]
  MoveL 2536 to (323.9, 11.48, -159.72) mm, rotated rx -179.9 ry 0 rz -90 deg; joints [37.105, -64.709, 102.995, -128.591, 50.504, 142.363]
  MoveL 2537 to (324.87, 11.41, -157.76) mm, rotated rx -179.9 ry 0 rz -90 deg; joints [37.183, -64.766, 103.083, -128.532, 50.571, 142.345]
  MoveL 2538 to (325.08, 11.33, -155.59) mm, rotated rx -179.9 ry 0 rz -90 deg; joints [37.242, -64.86, 103.227, -128.504, 50.638, 142.358]
  MoveL 2539 to (324.49, 11.25, -153.48) mm, rotated rx -179.9 ry 0 rz -90 deg; joints [37.274, -64.979, 103.409, -128.51, 50.697, 142.401]
  MoveL 2540 to (323.2, 11.18, -151.72) mm, rotated rx -179.9 ry 0 rz -90 deg; joints [37.275, -65.107, 103.604, -128.552, 50.74, 142.468]
  MoveL 2541 to (321.36, 11.1, -150.54) mm, rotated rx -179.9 ry 0 rz -90 deg; joints [37.246, -65.227, 103.787, -128.623, 50.761, 142.55]
  MoveL 2542 to (319.22, 11.02, -150.09) mm, rotated rx -179.9 ry 0 rz -90 deg; joints [37.189, -65.323, 103.935, -128.714, 50.759, 142.639]
  MoveL 2543 to (317.06, 10.95, -150.43) mm, rotated rx -179.9 ry 0 rz -90 deg; joints [37.112, -65.382, 104.029, -128.816, 50.735, 142.723]
  MoveL 2544 to (315.16, 10.87, -151.52) mm, rotated rx -179.9 ry 0 rz -90 deg; joints [37.026, -65.395, 104.057, -128.913, 50.691, 142.793]
  MoveL 2545 to (313.78, 10.79, -153.21) mm, rotated rx -179.9 ry 0 rz -90 deg; joints [36.941, -65.361, 104.015, -128.995, 50.634, 142.838]
  MoveL 2546 to (313.09, 10.72, -155.29) mm, rotated rx -179.9 ry 0 rz -90 deg; joints [36.869, -65.283, 103.909, -129.051, 50.573, 142.855]
  MoveL 2547 to (313.19, 10.64, -157.47) mm, rotated rx -179.9 ry 0 rz -90 deg; joints [36.82, -65.173, 103.753, -129.073, 50.515, 142.841]
  MoveL 2548 to (314.06, 10.56, -159.48) mm, rotated rx -179.9 ry 0 rz -90 deg; joints [36.8, -65.043, 103.569, -129.058, 50.468, 142.799]
  MoveL 2549 to (315.58, 10.49, -161.04) mm, rotated rx -179.9 ry 0 rz -90 deg; joints [36.811, -64.911, 103.38, -129.01, 50.438, 142.734]
  MoveL 2550 to (317.57, 10.41, -161.96) mm, rotated rx -179.9 ry 0 rz -90 deg; joints [36.852, -64.794, 103.212, -128.935, 50.431, 142.656]
  MoveL 2551 to (319.75, 10.33, -162.11) mm, rotated rx -179.9 ry 0 rz -90 deg; joints [36.917, -64.707, 103.087, -128.843, 50.448, 142.577]
  MoveL 2552 to (321.84, 10.26, -161.48) mm, rotated rx -179.9 ry 0 rz -90 deg; joints [36.999, -64.661, 103.022, -128.748, 50.486, 142.506]
  MoveL 2553 to (323.57, 10.18, -160.14) mm, rotated rx -179.9 ry 0 rz -90 deg; joints [37.085, -64.661, 103.025, -128.662, 50.541, 142.455]
  MoveL 2554 to (324.7, 10.1, -158.27) mm, rotated rx -179.9 ry 0 rz -90 deg; joints [37.166, -64.707, 103.098, -128.596, 50.607, 142.43]
  MoveL 2555 to (325.1, 10.02, -156.12) mm, rotated rx -179.9 ry 0 rz -90 deg; joints [37.23, -64.793, 103.23, -128.56, 50.675, 142.436]
  MoveL 2556 to (325.1, 10.02, -1) mm, rotated rx -179.9 ry 0 rz -90 deg; joints [41.302, -71.971, 113.318, -126.261, 54.923, 142.954]
  MoveL 2557 to (-325.1, 10.02, -1) mm, rotated rx -179.9 ry 0 rz -90 deg; joints [12.699, -90.932, 135.897, -162.037, 45.441, 167.607]
  MoveL 2558 to (-325.1, 10.02, -311.23) mm, rotated rx -179.9 ry 0 rz -90 deg; joints [9.724, -71.781, 113.658, -165.349, 41.872, 169.356]
  MoveL 2559 to (325.1, 10.03, -311.23) mm, rotated rx -179.9 ry 0 rz -90 deg; joints [33.798, -57.085, 91.451, -129.327, 45.968, 140.525]
  MoveL 2560 to (325.1, 10.02, -156.12) mm, rotated rx -179.9 ry 0 rz -90 deg; joints [37.23, -64.793, 103.23, -128.56, 50.675, 142.436]
  MoveC 2561 to (323.81, 10.03, -151.87) mm, rotated rx -179.9 ry 0 rz -90 deg; joints [37.292, -65.042, 103.596, -128.572, 50.786, 142.516] to (320.39, 10.03, -149.05) mm, rotated rx -179.9 ry 0 rz -90 deg; joints [37.252, -65.299, 103.976, -128.691, 50.838, 142.665]
  MoveL 2562 to (320.39, 10.02, -149.05) mm, rotated rx -179.9 ry 0 rz -90 deg; joints [37.252, -65.299, 103.976, -128.691, 50.838, 142.665]
  MoveC 2563 to (316.96, 10.02, -146.23) mm, rotated rx -179.9 ry 0 rz -90 deg; joints [37.211, -65.556, 104.355, -128.81, 50.89, 142.813] to (315.68, 10.02, -141.98) mm, rotated rx -179.9 ry 0 rz -90 deg; joints [37.273, -65.804, 104.717, -128.819, 50.999, 142.888]
  MoveL 2564 to (315.68, 10.03, -141.98) mm, rotated rx -179.9 ry 0 rz -90 deg; joints [37.273, -65.804, 104.717, -128.819, 50.999, 142.888]
  MoveL 2565 to (315.68, 10.02, -14.28) mm, rotated rx -179.9 ry 0 rz -90 deg; joints [40.618, -71.736, 113.016, -126.891, 54.471, 143.263]
  MoveC 2566 to (314.55, 10.03, -11.55) mm, rotated rx -179.9 ry 0 rz -90 deg; joints [40.658, -71.903, 113.242, -126.885, 54.53, 143.299] to (311.82, 10.02, -10.43) mm, rotated rx -179.9 ry 0 rz -90 deg; joints [40.6, -72.059, 113.455, -126.974, 54.53, 143.387]
  MoveL 2567 to (311.82, 10.02, -10.43) mm, rotated rx -179.9 ry 0 rz -90 deg; joints [40.6, -72.059, 113.455, -126.974, 54.53, 143.387]
  MoveL 2568 to (-311.82, 10.02, -10.43) mm, rotated rx -179.9 ry 0 rz -90 deg; joints [13.303, -90.1, 135.083, -161.218, 45.593, 167.047]
  MoveC 2569 to (-314.55, 10.03, -11.55) mm, rotated rx -179.9 ry 0 rz -90 deg; joints [13.141, -90.067, 135.052, -161.439, 45.558, 167.2] to (-315.68, 10.02, -14.28) mm, rotated rx -179.9 ry 0 rz -90 deg; joints [13.046, -89.904, 134.893, -161.571, 45.541, 167.291]
  MoveL 2570 to (-315.68, 10.02, -14.28) mm, rotated rx -179.9 ry 0 rz -90 deg; joints [13.046, -89.904, 134.893, -161.571, 45.541, 167.291]
  MoveL 2571 to (-315.68, 10.02, -297.96) mm, rotated rx -179.9 ry 0 rz -90 deg; joints [10.228, -72.463, 114.573, -164.677, 42.193, 168.905]
  MoveC 2572 to (-314.55, 10.02, -300.68) mm, rotated rx -179.9 ry 0 rz -90 deg; joints [10.255, -72.292, 114.342, -164.62, 42.141, 168.853] to (-311.82, 10.02, -301.81) mm, rotated rx -179.9 ry 0 rz -90 deg; joints [10.363, -72.197, 114.213, -164.452, 42.129, 168.724]
  MoveL 2573 to (-311.82, 10.03, -301.81) mm, rotated rx -179.9 ry 0 rz -90 deg; joints [10.363, -72.197, 114.213, -164.452, 42.129, 168.724]
  MoveL 2574 to (311.82, 10.03, -301.81) mm, rotated rx -179.9 ry 0 rz -90 deg; joints [33.585, -58.029, 92.956, -129.971, 46.191, 141.279]
  MoveC 2575 to (314.55, 10.03, -300.68) mm, rotated rx -179.9 ry 0 rz -90 deg; joints [33.692, -57.994, 92.899, -129.839, 46.244, 141.178] to (315.68, 10.02, -297.96) mm, rotated rx -179.9 ry 0 rz -90 deg; joints [33.782, -58.096, 93.058, -129.784, 46.337, 141.173]
  MoveL 2576 to (315.68, 10.02, -297.96) mm, rotated rx -179.9 ry 0 rz -90 deg; joints [33.782, -58.096, 93.058, -129.784, 46.337, 141.173]
  MoveL 2577 to (315.68, 10.03, -141.98) mm, rotated rx -179.9 ry 0 rz -90 deg; joints [37.273, -65.804, 104.717, -128.819, 50.999, 142.888]
  MoveC 2578 to (314.4, 10.03, -137.76) mm, rotated rx -179.9 ry 0 rz -90 deg; joints [37.336, -66.051, 105.076, -128.826, 51.107, 142.962] to (311, 10.02, -134.96) mm, rotated rx -179.9 ry 0 rz -90 deg; joints [37.295, -66.306, 105.449, -128.941, 51.156, 143.105]
  MoveL 2579 to (311, 10.02, -134.96) mm, rotated rx -179.9 ry 0 rz -90 deg; joints [37.295, -66.306, 105.449, -128.941, 51.156, 143.105]
  MoveC 2580 to (307.59, 10.02, -132.16) mm, rotated rx -179.9 ry 0 rz -90 deg; joints [37.255, -66.561, 105.821, -129.055, 51.205, 143.246] to (306.32, 10.02, -127.94) mm, rotated rx -179.9 ry 0 rz -90 deg; joints [37.317, -66.807, 106.176, -129.059, 51.312, 143.316]
  MoveL 2581 to (306.31, 10.02, -127.94) mm, rotated rx -179.9 ry 0 rz -90 deg; joints [37.317, -66.807, 106.176, -129.059, 51.312, 143.316]
  MoveL 2582 to (306.32, 10.02, -23.64) mm, rotated rx -179.9 ry 0 rz -90 deg; joints [40.049, -71.667, 112.936, -127.445, 54.124, 143.571]
  MoveC 2583 to (305.19, 10.03, -20.92) mm, rotated rx -179.9 ry 0 rz -90 deg; joints [40.088, -71.834, 113.163, -127.441, 54.183, 143.607] to (302.46, 10.03, -19.79) mm, rotated rx -179.9 ry 0 rz -90 deg; joints [40.029, -71.989, 113.375, -127.532, 54.183, 143.696]
  MoveL 2584 to (302.46, 10.03, -19.79) mm, rotated rx -179.9 ry 0 rz -90 deg; joints [40.029, -71.989, 113.375, -127.532, 54.183, 143.696]
  MoveL 2585 to (-302.46, 10.02, -19.79) mm, rotated rx -179.9 ry 0 rz -90 deg; joints [13.684, -89.336, 134.324, -160.701, 45.686, 166.693]
  MoveC 2586 to (-305.19, 10.02, -20.92) mm, rotated rx -179.9 ry 0 rz -90 deg; joints [13.524, -89.304, 134.294, -160.919, 45.65, 166.843] to (-306.32, 10.03, -23.64) mm, rotated rx -179.9 ry 0 rz -90 deg; joints [13.429, -89.143, 134.134, -161.049, 45.63, 166.933]
  MoveL 2587 to (-306.32, 10.02, -23.64) mm, rotated rx -179.9 ry 0 rz -90 deg; joints [13.429, -89.143, 134.134, -161.049, 45.63, 166.933]
  MoveL 2588 to (-306.32, 10.02, -288.59) mm, rotated rx -179.9 ry 0 rz -90 deg; joints [10.707, -72.912, 115.168, -164.024, 42.429, 168.456]
  MoveC 2589 to (-305.19, 10.02, -291.32) mm, rotated rx -179.9 ry 0 rz -90 deg; joints [10.733, -72.74, 114.938, -163.968, 42.378, 168.405] to (-302.46, 10.02, -292.45) mm, rotated rx -179.9 ry 0 rz -90 deg; joints [10.841, -72.644, 114.808, -163.801, 42.368, 168.277]
  MoveL 2590 to (-302.46, 10.03, -292.45) mm, rotated rx -179.9 ry 0 rz -90 deg; joints [10.841, -72.644, 114.808, -163.801, 42.368, 168.277]
  MoveL 2591 to (302.46, 10.02, -292.45) mm, rotated rx -179.9 ry 0 rz -90 deg; joints [33.489, -58.829, 94.22, -130.413, 46.43, 141.84]
  MoveC 2592 to (305.19, 10.02, -291.32) mm, rotated rx -179.9 ry 0 rz -90 deg; joints [33.596, -58.795, 94.164, -130.281, 46.483, 141.738] to (306.32, 10.02, -288.59) mm, rotated rx -179.9 ry 0 rz -90 deg; joints [33.687, -58.897, 94.322, -130.223, 46.575, 141.731]
  MoveL 2593 to (306.32, 10.03, -288.59) mm, rotated rx -179.9 ry 0 rz -90 deg; joints [33.687, -58.897, 94.322, -130.223, 46.575, 141.731]
  MoveL 2594 to (306.31, 10.02, -127.94) mm, rotated rx -179.9 ry 0 rz -90 deg; joints [37.317, -66.807, 106.176, -129.059, 51.312, 143.316]
  MoveC 2595 to (305.04, 10.03, -123.72) mm, rotated rx -179.9 ry 0 rz -90 deg; joints [37.38, -67.053, 106.529, -129.061, 51.417, 143.384] to (301.63, 10.03, -120.92) mm, rotated rx -179.9 ry 0 rz -90 deg; joints [37.34, -67.308, 106.898, -129.173, 51.464, 143.521]
  MoveL 2596 to (301.63, 10.02, -120.92) mm, rotated rx -179.9 ry 0 rz -90 deg; joints [37.34, -67.308, 106.898, -129.173, 51.464, 143.521]
  MoveC 2597 to (298.23, 10.02, -118.11) mm, rotated rx -179.9 ry 0 rz -90 deg; joints [37.299, -67.562, 107.264, -129.284, 51.511, 143.658] to (296.95, 10.02, -113.9) mm, rotated rx -179.9 ry 0 rz -90 deg; joints [37.362, -67.808, 107.615, -129.283, 51.615, 143.722]
  MoveL 2598 to (296.95, 10.02, -113.9) mm, rotated rx -179.9 ry 0 rz -90 deg; joints [37.362, -67.808, 107.615, -129.283, 51.615, 143.722]
  MoveL 2599 to (296.95, 10.03, -33) mm, rotated rx -179.9 ry 0 rz -90 deg; joints [39.481, -71.59, 112.845, -128.002, 53.777, 143.88]
  MoveC 2600 to (295.82, 10.03, -30.28) mm, rotated rx -179.9 ry 0 rz -90 deg; joints [39.518, -71.758, 113.073, -128, 53.836, 143.917] to (293.1, 10.03, -29.15) mm, rotated rx -179.9 ry 0 rz -90 deg; joints [39.459, -71.912, 113.284, -128.092, 53.836, 144.007]
  MoveL 2601 to (293.1, 10.02, -29.15) mm, rotated rx -179.9 ry 0 rz -90 deg; joints [39.459, -71.912, 113.284, -128.092, 53.836, 144.007]
  MoveL 2602 to (-293.1, 10.03, -29.15) mm, rotated rx -179.9 ry 0 rz -90 deg; joints [14.058, -88.575, 133.556, -160.192, 45.767, 166.342]
  MoveC 2603 to (-295.82, 10.02, -30.28) mm, rotated rx -179.9 ry 0 rz -90 deg; joints [13.899, -88.545, 133.527, -160.407, 45.731, 166.49] to (-296.95, 10.03, -33) mm, rotated rx -179.9 ry 0 rz -90 deg; joints [13.804, -88.386, 133.367, -160.536, 45.707, 166.578]
  MoveL 2604 to (-296.95, 10.03, -33) mm, rotated rx -179.9 ry 0 rz -90 deg; joints [13.804, -88.386, 133.367, -160.536, 45.707, 166.578]
  MoveL 2605 to (-296.95, 10.02, -279.23) mm, rotated rx -179.9 ry 0 rz -90 deg; joints [11.191, -73.356, 115.752, -163.367, 42.664, 168.007]
  MoveC 2606 to (-295.82, 10.03, -281.95) mm, rotated rx -179.9 ry 0 rz -90 deg; joints [11.216, -73.184, 115.523, -163.313, 42.615, 167.956] to (-293.1, 10.03, -283.08) mm, rotated rx -179.9 ry 0 rz -90 deg; joints [11.324, -73.086, 115.392, -163.146, 42.606, 167.829]
  MoveL 2607 to (-293.1, 10.03, -283.08) mm, rotated rx -179.9 ry 0 rz -90 deg; joints [11.324, -73.086, 115.392, -163.146, 42.606, 167.829]
  MoveL 2608 to (293.1, 10.02, -283.08) mm, rotated rx -179.9 ry 0 rz -90 deg; joints [33.391, -59.625, 95.468, -130.845, 46.664, 142.383]
  MoveC 2609 to (295.82, 10.02, -281.95) mm, rotated rx -179.9 ry 0 rz -90 deg; joints [33.499, -59.591, 95.413, -130.712, 46.716, 142.282] to (296.95, 10.03, -279.23) mm, rotated rx -179.9 ry 0 rz -90 deg; joints [33.591, -59.693, 95.568, -130.651, 46.808, 142.272]
  MoveL 2610 to (296.95, 10.02, -279.23) mm, rotated rx -179.9 ry 0 rz -90 deg; joints [33.591, -59.693, 95.568, -130.651, 46.808, 142.272]
  MoveL 2611 to (296.95, 10.02, -113.9) mm, rotated rx -179.9 ry 0 rz -90 deg; joints [37.362, -67.808, 107.615, -129.283, 51.615, 143.722]
  MoveC 2612 to (295.67, 10.02, -109.68) mm, rotated rx -179.9 ry 0 rz -90 deg; joints [37.426, -68.054, 107.964, -129.281, 51.719, 143.784] to (292.27, 10.02, -106.87) mm, rotated rx -179.9 ry 0 rz -90 deg; joints [37.385, -68.308, 108.327, -129.389, 51.763, 143.917]
  MoveL 2613 to (292.27, 10.02, -106.87) mm, rotated rx -179.9 ry 0 rz -90 deg; joints [37.385, -68.308, 108.327, -129.389, 51.763, 143.917]
  MoveC 2614 to (288.87, 10.03, -104.07) mm, rotated rx -179.9 ry 0 rz -90 deg; joints [37.344, -68.563, 108.689, -129.497, 51.807, 144.048] to (287.59, 10.02, -99.85) mm, rotated rx -179.9 ry 0 rz -90 deg; joints [37.408, -68.808, 109.035, -129.492, 51.909, 144.107]
  MoveL 2615 to (287.59, 10.02, -99.85) mm, rotated rx -179.9 ry 0 rz -90 deg; joints [37.408, -68.808, 109.035, -129.492, 51.909, 144.107]
  MoveL 2616 to (287.59, 10.02, -42.37) mm, rotated rx -179.9 ry 0 rz -90 deg; joints [38.914, -71.505, 112.744, -128.561, 53.432, 144.192]
  MoveC 2617 to (286.46, 10.02, -39.64) mm, rotated rx -179.9 ry 0 rz -90 deg; joints [38.95, -71.674, 112.973, -128.56, 53.491, 144.23] to (283.74, 10.03, -38.51) mm, rotated rx -179.9 ry 0 rz -90 deg; joints [38.889, -71.827, 113.183, -128.654, 53.491, 144.32]
  MoveL 2618 to (283.74, 10.03, -38.51) mm, rotated rx -179.9 ry 0 rz -90 deg; joints [38.889, -71.827, 113.183, -128.654, 53.491, 144.32]
  MoveL 2619 to (-283.74, 10.02, -38.51) mm, rotated rx -179.9 ry 0 rz -90 deg; joints [14.423, -87.818, 132.779, -159.691, 45.837, 165.994]
  MoveC 2620 to (-286.46, 10.02, -39.64) mm, rotated rx -179.9 ry 0 rz -90 deg; joints [14.266, -87.79, 132.752, -159.904, 45.8, 166.14] to (-287.59, 10.03, -42.37) mm, rotated rx -179.9 ry 0 rz -90 deg; joints [14.171, -87.633, 132.591, -160.031, 45.773, 166.226]
  MoveL 2621 to (-287.59, 10.02, -42.37) mm, rotated rx -179.9 ry 0 rz -90 deg; joints [14.171, -87.633, 132.591, -160.031, 45.773, 166.226]
  MoveL 2622 to (-287.59, 10.02, -269.87) mm, rotated rx -179.9 ry 0 rz -90 deg; joints [11.68, -73.795, 116.326, -162.706, 42.898, 167.556]
  MoveC 2623 to (-286.46, 10.02, -272.59) mm, rotated rx -179.9 ry 0 rz -90 deg; joints [11.704, -73.622, 116.098, -162.653, 42.851, 167.507] to (-283.74, 10.02, -273.72) mm, rotated rx -179.9 ry 0 rz -90 deg; joints [11.812, -73.524, 115.966, -162.488, 42.843, 167.381]
  MoveL 2624 to (-283.74, 10.02, -273.72) mm, rotated rx -179.9 ry 0 rz -90 deg; joints [11.812, -73.524, 115.966, -162.488, 42.843, 167.381]
  MoveL 2625 to (283.74, 10.02, -273.72) mm, rotated rx -179.9 ry 0 rz -90 deg; joints [33.291, -60.416, 96.699, -131.265, 46.892, 142.912]
  MoveC 2626 to (286.46, 10.03, -272.59) mm, rotated rx -179.9 ry 0 rz -90 deg; joints [33.4, -60.383, 96.645, -131.131, 46.944, 142.811] to (287.59, 10.02, -269.87) mm, rotated rx -179.9 ry 0 rz -90 deg; joints [33.492, -60.484, 96.799, -131.068, 47.035, 142.798]
  MoveL 2627 to (287.59, 10.02, -269.87) mm, rotated rx -179.9 ry 0 rz -90 deg; joints [33.492, -60.484, 96.799, -131.068, 47.035, 142.798]
  MoveL 2628 to (287.59, 10.02, -99.85) mm, rotated rx -179.9 ry 0 rz -90 deg; joints [37.408, -68.808, 109.035, -129.492, 51.909, 144.107]
  MoveC 2629 to (286.31, 10.03, -95.63) mm, rotated rx -179.9 ry 0 rz -90 deg; joints [37.473, -69.054, 109.38, -129.485, 52.01, 144.164] to (282.91, 10.02, -92.83) mm, rotated rx -179.9 ry 0 rz -90 deg; joints [37.432, -69.308, 109.739, -129.591, 52.052, 144.292]
  MoveL 2630 to (282.91, 10.02, -92.83) mm, rotated rx -179.9 ry 0 rz -90 deg; joints [37.432, -69.308, 109.739, -129.591, 52.052, 144.292]
  MoveC 2631 to (279.5, 10.03, -90.03) mm, rotated rx -179.9 ry 0 rz -90 deg; joints [37.39, -69.563, 110.096, -129.695, 52.094, 144.418] to (278.23, 10.03, -85.81) mm, rotated rx -179.9 ry 0 rz -90 deg; joints [37.456, -69.808, 110.438, -129.685, 52.193, 144.471]
  MoveL 2632 to (278.23, 10.03, -85.81) mm, rotated rx -179.9 ry 0 rz -90 deg; joints [37.456, -69.808, 110.438, -129.685, 52.193, 144.471]
  MoveL 2633 to (278.23, 10.02, -51.73) mm, rotated rx -179.9 ry 0 rz -90 deg; joints [38.348, -71.413, 112.632, -129.122, 53.088, 144.506]
  MoveC 2634 to (277.1, 10.03, -49.01) mm, rotated rx -179.9 ry 0 rz -90 deg; joints [38.383, -71.582, 112.862, -129.122, 53.147, 144.544] to (274.37, 10.03, -47.88) mm, rotated rx -179.9 ry 0 rz -90 deg; joints [38.321, -71.735, 113.071, -129.217, 53.147, 144.635]
  MoveL 2635 to (274.37, 10.03, -47.88) mm, rotated rx -179.9 ry 0 rz -90 deg; joints [38.321, -71.735, 113.071, -129.217, 53.147, 144.635]
  MoveL 2636 to (-274.37, 10.03, -47.88) mm, rotated rx -179.9 ry 0 rz -90 deg; joints [14.78, -87.065, 131.994, -159.198, 45.896, 165.648]
  MoveC 2637 to (-277.1, 10.03, -49.01) mm, rotated rx -179.9 ry 0 rz -90 deg; joints [14.625, -87.038, 131.967, -159.408, 45.858, 165.792] to (-278.23, 10.02, -51.73) mm, rotated rx -179.9 ry 0 rz -90 deg; joints [14.53, -86.883, 131.806, -159.533, 45.829, 165.876]
  MoveL 2638 to (-278.23, 10.02, -51.73) mm, rotated rx -179.9 ry 0 rz -90 deg; joints [14.53, -86.883, 131.806, -159.533, 45.829, 165.876]
  MoveL 2639 to (-278.23, 10.02, -260.51) mm, rotated rx -179.9 ry 0 rz -90 deg; joints [12.175, -74.23, 116.89, -162.041, 43.132, 167.105]
  MoveC 2640 to (-277.1, 10.02, -263.23) mm, rotated rx -179.9 ry 0 rz -90 deg; joints [12.198, -74.056, 116.662, -161.99, 43.086, 167.057] to (-274.37, 10.02, -264.36) mm, rotated rx -179.9 ry 0 rz -90 deg; joints [12.306, -73.956, 116.529, -161.825, 43.079, 166.931]
  MoveL 2641 to (-274.37, 10.03, -264.36) mm, rotated rx -179.9 ry 0 rz -90 deg; joints [12.306, -73.956, 116.529, -161.825, 43.079, 166.931]
